LIN {X 0,Y 574.396,Z 596.267,A -85,B 0,C 180,E1 -2267.811,E2 -2267.811} C_VEL
LIN {X 0,Y 574.661,Z 582.717,A -85,B 0,C 180,E1 -2268.633,E2 -2268.633} C_VEL
LIN {X 0,Y 574.868,Z 568.152,A -85,B 0,C 180,E1 -2269.364,E2 -2269.364} C_VEL
LIN {X 0,Y 575.125,Z 552.245,A -85,B 0,C 180,E1 -2270.008,E2 -2270.008} C_VEL
LIN {X 0,Y 575.36,Z 536.014,A -85,B 0,C 180,E1 -2270.513,E2 -2270.513} C_VEL
LIN {X 0,Y 575.491,Z 519.437,A -85,B 0,C 180,E1 -2270.882,E2 -2270.882} C_VEL
LIN {X 0,Y 576.152,Z 335.908,A -85,B 0,C 180,E1 -2273.297,E2 -2273.297} C_VEL
LIN {X 0,Y 576.125,Z 317.842,A -85,B 0,C 180,E1 -2273.539,E2 -2273.539} C_VEL
LIN {X 0,Y 575.045,Z 311.76,A -85,B 0,C 180,E1 -2273.688,E2 -2273.688} C_VEL
LIN {X 0,Y 575.605,Z 275.988,A -85,B 0,C 180,E1 -2276.796,E2 -2276.796} C_VEL
LIN {X 0,Y 575.443,Z 270.866,A -85,B 0,C 180,E1 -2277.257,E2 -2277.257} C_VEL
LIN {X 0,Y 573.255,Z 263.39,A -85,B 0,C 180,E1 -2278.04,E2 -2278.04} C_VEL
LIN {X 0,Y 573.23,Z 263.394,A -85,B 0,C 180,E1 -2280.883,E2 -2280.883} C_VEL
LIN {X 0,Y 573.26,Z 263.392,A -85,B 0,C 180,E1 -2283.524,E2 -2283.524} C_VEL
LIN {X 0,Y 573.213,Z 263.391,A -85,B 0,C 180,E1 -2286.051,E2 -2286.051} C_VEL
LIN {X 0,Y 573.245,Z 263.388,A -85,B 0,C 180,E1 -2288.701,E2 -2288.701} C_VEL
LIN {X 0,Y 573.251,Z 263.39,A -85,B 0,C 180,E1 -2291.595,E2 -2291.595} C_VEL
LIN {X 0,Y 573.237,Z 263.387,A -85,B 0,C 180,E1 -2294.333,E2 -2294.333} C_VEL
LIN {X 0,Y 573.237,Z 263.394,A -85,B 0,C 180,E1 -2297.358,E2 -2297.358} C_VEL
LIN {X 0,Y 573.272,Z 263.388,A -85,B 0,C 180,E1 -2299.477,E2 -2299.477} C_VEL
LIN {X 0,Y 573.233,Z 263.387,A -85,B 0,C 180,E1 -2302.192,E2 -2302.192} C_VEL
LIN {X 0,Y 573.253,Z 263.388,A -85,B 0,C 180,E1 -2304.816,E2 -2304.816} C_VEL
LIN {X 0,Y 573.25,Z 263.393,A -85,B 0,C 180,E1 -2307.355,E2 -2307.355} C_VEL
LIN {X 0,Y 573.245,Z 263.386,A -85,B 0,C 180,E1 -2310.512,E2 -2310.512} C_VEL
LIN {X 0,Y 573.247,Z 263.393,A -85,B 0,C 180,E1 -2313.024,E2 -2313.024} C_VEL
LIN {X 0,Y 573.272,Z 263.389,A -85,B 0,C 180,E1 -2315.366,E2 -2315.366} C_VEL
LIN {X 0,Y 573.226,Z 263.389,A -85,B 0,C 180,E1 -2318.419,E2 -2318.419} C_VEL
LIN {X 0,Y 573.266,Z 263.383,A -85,B 0,C 180,E1 -2320.731,E2 -2320.731} C_VEL
LIN {X 0,Y 573.248,Z 263.388,A -85,B 0,C 180,E1 -2323.622,E2 -2323.622} C_VEL
LIN {X 0,Y 573.27,Z 263.38,A -85,B 0,C 180,E1 -2325.807,E2 -2325.807} C_VEL
LIN {X 0,Y 573.26,Z 263.387,A -85,B 0,C 180,E1 -2328.745,E2 -2328.745} C_VEL
LIN {X 0,Y 573.282,Z 263.383,A -85,B 0,C 180,E1 -2331.541,E2 -2331.541} C_VEL
LIN {X 0,Y 573.295,Z 263.377,A -85,B 0,C 180,E1 -2334.372,E2 -2334.372} C_VEL
LIN {X 0,Y 573.312,Z 263.378,A -85,B 0,C 180,E1 -2337.893,E2 -2337.893} C_VEL
LIN {X 0,Y 573.327,Z 263.377,A -85,B 0,C 180,E1 -2340.702,E2 -2340.702} C_VEL
LIN {X 0,Y 573.302,Z 263.383,A -85,B 0,C 180,E1 -2342.811,E2 -2342.811} C_VEL
LIN {X 0,Y 573.295,Z 263.38,A -85,B 0,C 180,E1 -2345.628,E2 -2345.628} C_VEL
LIN {X 0,Y 573.282,Z 263.379,A -85,B 0,C 180,E1 -2348.46,E2 -2348.46} C_VEL
LIN {X 0,Y 573.27,Z 263.388,A -85,B 0,C 180,E1 -2351.312,E2 -2351.312} C_VEL
LIN {X 0,Y 573.28,Z 263.382,A -85,B 0,C 180,E1 -2354.425,E2 -2354.425} C_VEL
LIN {X 0,Y 573.256,Z 263.392,A -85,B 0,C 180,E1 -2357.112,E2 -2357.112} C_VEL
LIN {X 0,Y 573.249,Z 263.385,A -85,B 0,C 180,E1 -2360.077,E2 -2360.077} C_VEL
LIN {X 0,Y 573.232,Z 263.395,A -85,B 0,C 180,E1 -2363.1,E2 -2363.1} C_VEL
LIN {X 0,Y 573.248,Z 263.387,A -85,B 0,C 180,E1 -2364.383,E2 -2364.383} C_VEL
LIN {X 0,Y 572.621,Z 263.473,A -85,B 0,C 180,E1 -2364.97,E2 -2364.97} C_VEL
LIN {X 0,Y 569.779,Z 263.826,A -85,B 0,C 180,E1 -2365.921,E2 -2365.921} C_VEL
LIN {X 0,Y 567.347,Z 264.127,A -85,B 0,C 180,E1 -2366.686,E2 -2366.686} C_VEL
LIN {X 0,Y 566.292,Z 264.253,A -85,B 0,C 180,E1 -2367.277,E2 -2367.277} C_VEL
LIN {X 0,Y 566.201,Z 264.261,A -85,B 0,C 180,E1 -2367.478,E2 -2367.478} C_VEL
LIN {X 0,Y 566.199,Z 264.264,A -85,B 0,C 180,E1 -2369.769,E2 -2369.769} C_VEL
LIN {X 0,Y 566.201,Z 264.266,A -85,B 0,C 180,E1 -2372.43,E2 -2372.43} C_VEL
LIN {X 0,Y 566.212,Z 264.27,A -85,B 0,C 180,E1 -2374.995,E2 -2374.995} C_VEL
LIN {X 0,Y 566.195,Z 264.263,A -85,B 0,C 180,E1 -2377.461,E2 -2377.461} C_VEL
LIN {X 0,Y 566.206,Z 264.264,A -85,B 0,C 180,E1 -2380.199,E2 -2380.199} C_VEL
LIN {X 0,Y 566.2,Z 264.27,A -85,B 0,C 180,E1 -2383.054,E2 -2383.054} C_VEL
LIN {X 0,Y 566.201,Z 264.262,A -85,B 0,C 180,E1 -2386.049,E2 -2386.049} C_VEL
LIN {X 0,Y 566.211,Z 264.272,A -85,B 0,C 180,E1 -2388.864,E2 -2388.864} C_VEL
LIN {X 0,Y 566.188,Z 264.264,A -85,B 0,C 180,E1 -2391.637,E2 -2391.637} C_VEL
LIN {X 0,Y 566.161,Z 264.27,A -85,B 0,C 180,E1 -2394.308,E2 -2394.308} C_VEL
LIN {X 0,Y 566.219,Z 264.266,A -85,B 0,C 180,E1 -2396.898,E2 -2396.898} C_VEL
LIN {X 0,Y 566.183,Z 264.269,A -85,B 0,C 180,E1 -2399.408,E2 -2399.408} C_VEL
LIN {X 0,Y 566.212,Z 264.265,A -85,B 0,C 180,E1 -2401.858,E2 -2401.858} C_VEL
LIN {X 0,Y 566.254,Z 264.454,A -85,B 0,C 180,E1 -2404.13,E2 -2404.13} C_VEL
LIN {X 0,Y 568.203,Z 272.217,A -85,B 0,C 180,E1 -2405.022,E2 -2405.022} C_VEL
LIN {X 0,Y 568.08,Z 282.889,A -85,B 0,C 180,E1 -2406.085,E2 -2406.085} C_VEL
LIN {X 0,Y 569.697,Z 291.686,A -85,B 0,C 180,E1 -2406.276,E2 -2406.276} C_VEL
LIN {X 0,Y 568.883,Z 488.854,A -85,B 0,C 180,E1 -2408.9,E2 -2408.9} C_VEL
LIN {X 0,Y 568.716,Z 505.193,A -85,B 0,C 180,E1 -2409.26,E2 -2409.26} C_VEL
LIN {X 0,Y 568.457,Z 521.005,A -85,B 0,C 180,E1 -2409.747,E2 -2409.747} C_VEL
LIN {X 0,Y 568.168,Z 537.348,A -85,B 0,C 180,E1 -2410.405,E2 -2410.405} C_VEL
LIN {X 0,Y 567.887,Z 551.932,A -85,B 0,C 180,E1 -2411.137,E2 -2411.137} C_VEL
LIN {X 0,Y 567.549,Z 566.935,A -85,B 0,C 180,E1 -2412.055,E2 -2412.055} C_VEL
LIN {X 0,Y 567.21,Z 580.823,A -85,B 0,C 180,E1 -2413.072,E2 -2413.072} C_VEL
LIN {X 0,Y 566.947,Z 593.594,A -85,B 0,C 180,E1 -2414.174,E2 -2414.174} C_VEL
LIN {X 0,Y 566.624,Z 605.25,A -85,B 0,C 180,E1 -2415.342,E2 -2415.342} C_VEL
LIN {X 0,Y 566.435,Z 617.002,A -85,B 0,C 180,E1 -2416.73,E2 -2416.73} C_VEL
LIN {X 0,Y 566.241,Z 627.369,A -85,B 0,C 180,E1 -2418.183,E2 -2418.183} C_VEL
LIN {X 0,Y 566.133,Z 636.034,A -85,B 0,C 180,E1 -2419.63,E2 -2419.63} C_VEL
LIN {X 0,Y 566.012,Z 643.287,A -85,B 0,C 180,E1 -2421.071,E2 -2421.071} C_VEL
LIN {X 0,Y 565.97,Z 649.294,A -85,B 0,C 180,E1 -2422.508,E2 -2422.508} C_VEL
LIN {X 0,Y 565.915,Z 654.055,A -85,B 0,C 180,E1 -2423.941,E2 -2423.941} C_VEL
LIN {X 0,Y 565.913,Z 658.544,A -85,B 0,C 180,E1 -2425.727,E2 -2425.727} C_VEL
LIN {X 0,Y 565.866,Z 661.021,A -85,B 0,C 180,E1 -2427.152,E2 -2427.152} C_VEL
LIN {X 0,Y 565.84,Z 662.45,A -85,B 0,C 180,E1 -2428.577,E2 -2428.577} C_VEL
LIN {X 0,Y 565.835,Z 662.996,A -85,B 0,C 180,E1 -2430,E2 -2430} C_VEL
LIN {X 0,Y 565.838,Z 662.509,A -85,B 0,C 180,E1 -2431.423,E2 -2431.423} C_VEL
LIN {X 0,Y 565.867,Z 661.149,A -85,B 0,C 180,E1 -2432.848,E2 -2432.848} C_VEL
LIN {X 0,Y 565.91,Z 658.728,A -85,B 0,C 180,E1 -2434.273,E2 -2434.273} C_VEL
LIN {X 0,Y 565.964,Z 655.378,A -85,B 0,C 180,E1 -2435.701,E2 -2435.701} C_VEL
LIN {X 0,Y 565.967,Z 650.873,A -85,B 0,C 180,E1 -2437.133,E2 -2437.133} C_VEL
LIN {X 0,Y 566.022,Z 645.304,A -85,B 0,C 180,E1 -2438.569,E2 -2438.569} C_VEL
LIN {X 0,Y 566.084,Z 638.461,A -85,B 0,C 180,E1 -2440.009,E2 -2440.009} C_VEL
LIN {X 0,Y 566.209,Z 630.214,A -85,B 0,C 180,E1 -2441.455,E2 -2441.455} C_VEL
LIN {X 0,Y 566.363,Z 620.389,A -85,B 0,C 180,E1 -2442.906,E2 -2442.906} C_VEL
LIN {X 0,Y 566.58,Z 610.288,A -85,B 0,C 180,E1 -2444.181,E2 -2444.181} C_VEL
LIN {X 0,Y 566.797,Z 598.38,A -85,B 0,C 180,E1 -2445.461,E2 -2445.461} C_VEL
LIN {X 0,Y 567.124,Z 585.297,A -85,B 0,C 180,E1 -2446.653,E2 -2446.653} C_VEL
LIN {X 0,Y 567.419,Z 572.581,A -85,B 0,C 180,E1 -2447.641,E2 -2447.641} C_VEL
LIN {X 0,Y 567.757,Z 558.218,A -85,B 0,C 180,E1 -2448.587,E2 -2448.587} C_VEL
LIN {X 0,Y 568.074,Z 543.006,A -85,B 0,C 180,E1 -2449.42,E2 -2449.42} C_VEL
LIN {X 0,Y 568.353,Z 528.125,A -85,B 0,C 180,E1 -2450.077,E2 -2450.077} C_VEL
LIN {X 0,Y 568.613,Z 512.384,A -85,B 0,C 180,E1 -2450.625,E2 -2450.625} C_VEL
LIN {X 0,Y 568.809,Z 495.094,A -85,B 0,C 180,E1 -2451.068,E2 -2451.068} C_VEL
LIN {X 0,Y 568.982,Z 478.408,A -85,B 0,C 180,E1 -2451.345,E2 -2451.345} C_VEL
LIN {X 0,Y 569.679,Z 290.701,A -85,B 0,C 180,E1 -2453.828,E2 -2453.828} C_VEL
LIN {X 0,Y 568.068,Z 282.675,A -85,B 0,C 180,E1 -2454.027,E2 -2454.027} C_VEL
LIN {X 0,Y 568.089,Z 271.64,A -85,B 0,C 180,E1 -2455.133,E2 -2455.133} C_VEL
LIN {X 0,Y 566.221,Z 264.268,A -85,B 0,C 180,E1 -2455.995,E2 -2455.995} C_VEL
LIN {X 0,Y 566.186,Z 264.272,A -85,B 0,C 180,E1 -2458.953,E2 -2458.953} C_VEL
LIN {X 0,Y 566.191,Z 264.274,A -85,B 0,C 180,E1 -2461.422,E2 -2461.422} C_VEL
LIN {X 0,Y 566.208,Z 264.266,A -85,B 0,C 180,E1 -2463.956,E2 -2463.956} C_VEL
LIN {X 0,Y 566.181,Z 264.264,A -85,B 0,C 180,E1 -2466.571,E2 -2466.571} C_VEL
LIN {X 0,Y 566.213,Z 264.266,A -85,B 0,C 180,E1 -2469.685,E2 -2469.685} C_VEL
LIN {X 0,Y 566.203,Z 264.267,A -85,B 0,C 180,E1 -2472.917,E2 -2472.917} C_VEL
LIN {X 0,Y 566.197,Z 264.264,A -85,B 0,C 180,E1 -2476.048,E2 -2476.048} C_VEL
LIN {X 0,Y 566.177,Z 264.27,A -85,B 0,C 180,E1 -2478.861,E2 -2478.861} C_VEL
LIN {X 0,Y 566.184,Z 264.268,A -85,B 0,C 180,E1 -2481.637,E2 -2481.637} C_VEL
LIN {X 0,Y 566.195,Z 264.264,A -85,B 0,C 180,E1 -2484.31,E2 -2484.31} C_VEL
LIN {X 0,Y 566.217,Z 264.266,A -85,B 0,C 180,E1 -2486.898,E2 -2486.898} C_VEL
LIN {X 0,Y 566.179,Z 264.272,A -85,B 0,C 180,E1 -2489.407,E2 -2489.407} C_VEL
LIN {X 0,Y 566.209,Z 264.26,A -85,B 0,C 180,E1 -2491.857,E2 -2491.857} C_VEL
LIN {X 0,Y 566.21,Z 264.262,A -85,B 0,C 180,E1 -2494.251,E2 -2494.251} C_VEL
LIN {X 0,Y 566.189,Z 264.268,A -85,B 0,C 180,E1 -2496.714,E2 -2496.714} C_VEL
LIN {X 0,Y 566.206,Z 264.265,A -85,B 0,C 180,E1 -2499.662,E2 -2499.662} C_VEL
LIN {X 0,Y 566.197,Z 264.267,A -85,B 0,C 180,E1 -2502.668,E2 -2502.668} C_VEL
LIN {X 0,Y 566.232,Z 264.261,A -85,B 0,C 180,E1 -2505.627,E2 -2505.627} C_VEL
LIN {X 0,Y 566.232,Z 264.263,A -85,B 0,C 180,E1 -2508.675,E2 -2508.675} C_VEL
LIN {X 0,Y 566.225,Z 264.263,A -85,B 0,C 180,E1 -2511.434,E2 -2511.434} C_VEL
LIN {X 0,Y 566.265,Z 264.256,A -85,B 0,C 180,E1 -2514.302,E2 -2514.302} C_VEL
LIN {X 0,Y 566.282,Z 264.25,A -85,B 0,C 180,E1 -2517.866,E2 -2517.866} C_VEL
LIN {X 0,Y 566.299,Z 264.257,A -85,B 0,C 180,E1 -2520.711,E2 -2520.711} C_VEL
LIN {X 0,Y 566.269,Z 264.262,A -85,B 0,C 180,E1 -2522.845,E2 -2522.845} C_VEL
LIN {X 0,Y 566.265,Z 264.256,A -85,B 0,C 180,E1 -2525.698,E2 -2525.698} C_VEL
LIN {X 0,Y 566.225,Z 264.264,A -85,B 0,C 180,E1 -2528.566,E2 -2528.566} C_VEL
LIN {X 0,Y 566.239,Z 264.26,A -85,B 0,C 180,E1 -2531.454,E2 -2531.454} C_VEL
LIN {X 0,Y 566.231,Z 264.263,A -85,B 0,C 180,E1 -2534.507,E2 -2534.507} C_VEL
LIN {X 0,Y 566.197,Z 264.267,A -85,B 0,C 180,E1 -2537.332,E2 -2537.332} C_VEL
LIN {X 0,Y 566.21,Z 264.265,A -85,B 0,C 180,E1 -2540.337,E2 -2540.337} C_VEL
LIN {X 0,Y 566.186,Z 264.268,A -85,B 0,C 180,E1 -2543.404,E2 -2543.404} C_VEL
LIN {X 0,Y 566.209,Z 264.263,A -85,B 0,C 180,E1 -2545.749,E2 -2545.749} C_VEL
LIN {X 0,Y 566.199,Z 264.266,A -85,B 0,C 180,E1 -2548.202,E2 -2548.202} C_VEL
LIN {X 0,Y 566.188,Z 264.272,A -85,B 0,C 180,E1 -2551.077,E2 -2551.077} C_VEL
LIN {X 0,Y 566.209,Z 264.264,A -85,B 0,C 180,E1 -2553.734,E2 -2553.734} C_VEL
LIN {X 0,Y 566.213,Z 264.269,A -85,B 0,C 180,E1 -2556.569,E2 -2556.569} C_VEL
LIN {X 0,Y 566.204,Z 264.264,A -85,B 0,C 180,E1 -2559.685,E2 -2559.685} C_VEL
LIN {X 0,Y 566.21,Z 264.265,A -85,B 0,C 180,E1 -2562.087,E2 -2562.087} C_VEL
LIN {X 0,Y 566.171,Z 264.273,A -85,B 0,C 180,E1 -2565.036,E2 -2565.036} C_VEL
LIN {X 0,Y 566.216,Z 264.264,A -85,B 0,C 180,E1 -2568.136,E2 -2568.136} C_VEL
LIN {X 0,Y 566.217,Z 264.271,A -85,B 0,C 180,E1 -2570.727,E2 -2570.727} C_VEL
LIN {X 0,Y 566.182,Z 264.267,A -85,B 0,C 180,E1 -2573.788,E2 -2573.788} C_VEL
LIN {X 0,Y 566.209,Z 264.264,A -85,B 0,C 180,E1 -2576.266,E2 -2576.266} C_VEL
LIN {X 0,Y 566.191,Z 264.273,A -85,B 0,C 180,E1 -2578.923,E2 -2578.923} C_VEL
LIN {X 0,Y 566.24,Z 264.409,A -85,B 0,C 180,E1 -2581.703,E2 -2581.703} C_VEL
LIN {X 0,Y 568.798,Z 273.135,A -85,B 0,C 180,E1 -2582.617,E2 -2582.617} C_VEL
LIN {X 0,Y 568.763,Z 287.404,A -85,B 0,C 180,E1 -2583.883,E2 -2583.883} C_VEL
LIN {X 0,Y 568.329,Z 311.996,A -85,B 0,C 180,E1 -2586.036,E2 -2586.036} C_VEL
LIN {X 0,Y 569.734,Z 319.846,A -85,B 0,C 180,E1 -2586.208,E2 -2586.208} C_VEL
LIN {X 0,Y 568.873,Z 519.439,A -85,B 0,C 180,E1 -2588.864,E2 -2588.864} C_VEL
LIN {X 0,Y 568.726,Z 536.014,A -85,B 0,C 180,E1 -2589.237,E2 -2589.237} C_VEL
LIN {X 0,Y 568.422,Z 552.246,A -85,B 0,C 180,E1 -2589.746,E2 -2589.746} C_VEL
LIN {X 0,Y 568.148,Z 568.383,A -85,B 0,C 180,E1 -2590.408,E2 -2590.408} C_VEL
LIN {X 0,Y 567.878,Z 582.718,A -85,B 0,C 180,E1 -2591.136,E2 -2591.136} C_VEL
LIN {X 0,Y 567.582,Z 596.271,A -85,B 0,C 180,E1 -2591.968,E2 -2591.968} C_VEL
LIN {X 0,Y 567.228,Z 610.22,A -85,B 0,C 180,E1 -2592.98,E2 -2592.98} C_VEL
LIN {X 0,Y 566.915,Z 624.071,A -85,B 0,C 180,E1 -2594.173,E2 -2594.173} C_VEL
LIN {X 0,Y 566.63,Z 635.62,A -85,B 0,C 180,E1 -2595.339,E2 -2595.339} C_VEL
LIN {X 0,Y 566.434,Z 647.338,A -85,B 0,C 180,E1 -2596.73,E2 -2596.73} C_VEL
LIN {X 0,Y 566.238,Z 657.673,A -85,B 0,C 180,E1 -2598.183,E2 -2598.183} C_VEL
LIN {X 0,Y 566.12,Z 666.285,A -85,B 0,C 180,E1 -2599.63,E2 -2599.63} C_VEL
LIN {X 0,Y 566.001,Z 673.489,A -85,B 0,C 180,E1 -2601.071,E2 -2601.071} C_VEL
LIN {X 0,Y 565.968,Z 679.467,A -85,B 0,C 180,E1 -2602.508,E2 -2602.508} C_VEL
LIN {X 0,Y 565.915,Z 684.187,A -85,B 0,C 180,E1 -2603.941,E2 -2603.941} C_VEL
LIN {X 0,Y 565.911,Z 688.637,A -85,B 0,C 180,E1 -2605.727,E2 -2605.727} C_VEL
LIN {X 0,Y 565.866,Z 691.089,A -85,B 0,C 180,E1 -2607.152,E2 -2607.152} C_VEL
LIN {X 0,Y 565.839,Z 692.48,A -85,B 0,C 180,E1 -2608.577,E2 -2608.577} C_VEL
LIN {X 0,Y 565.834,Z 693,A -85,B 0,C 180,E1 -2610,E2 -2610} C_VEL
LIN {X 0,Y 565.839,Z 692.48,A -85,B 0,C 180,E1 -2611.423,E2 -2611.423} C_VEL
LIN {X 0,Y 565.866,Z 691.088,A -85,B 0,C 180,E1 -2612.848,E2 -2612.848} C_VEL
LIN {X 0,Y 565.911,Z 688.636,A -85,B 0,C 180,E1 -2614.273,E2 -2614.273} C_VEL
LIN {X 0,Y 565.914,Z 684.188,A -85,B 0,C 180,E1 -2616.059,E2 -2616.059} C_VEL
LIN {X 0,Y 565.968,Z 679.468,A -85,B 0,C 180,E1 -2617.492,E2 -2617.492} C_VEL
LIN {X 0,Y 566.001,Z 673.489,A -85,B 0,C 180,E1 -2618.929,E2 -2618.929} C_VEL
LIN {X 0,Y 566.126,Z 665.277,A -85,B 0,C 180,E1 -2620.551,E2 -2620.551} C_VEL
LIN {X 0,Y 566.246,Z 656.443,A -85,B 0,C 180,E1 -2621.999,E2 -2621.999} C_VEL
LIN {X 0,Y 566.427,Z 645.908,A -85,B 0,C 180,E1 -2623.453,E2 -2623.453} C_VEL
LIN {X 0,Y 566.66,Z 634.612,A -85,B 0,C 180,E1 -2624.773,E2 -2624.773} C_VEL
LIN {X 0,Y 566.957,Z 622.119,A -85,B 0,C 180,E1 -2626.01,E2 -2626.01} C_VEL
LIN {X 0,Y 567.229,Z 609.046,A -85,B 0,C 180,E1 -2627.113,E2 -2627.113} C_VEL
LIN {X 0,Y 567.6,Z 594.852,A -85,B 0,C 180,E1 -2628.125,E2 -2628.125} C_VEL
LIN {X 0,Y 567.9,Z 581.028,A -85,B 0,C 180,E1 -2628.957,E2 -2628.957} C_VEL
LIN {X 0,Y 568.196,Z 566.527,A -85,B 0,C 180,E1 -2629.678,E2 -2629.678} C_VEL
LIN {X 0,Y 568.444,Z 550.945,A -85,B 0,C 180,E1 -2630.301,E2 -2630.301} C_VEL
LIN {X 0,Y 568.734,Z 534.187,A -85,B 0,C 180,E1 -2630.81,E2 -2630.81} C_VEL
LIN {X 0,Y 568.889,Z 517.947,A -85,B 0,C 180,E1 -2631.159,E2 -2631.159} C_VEL
LIN {X 0,Y 569.679,Z 320.023,A -85,B 0,C 180,E1 -2633.792,E2 -2633.792} C_VEL
LIN {X 0,Y 568.354,Z 311.826,A -85,B 0,C 180,E1 -2633.978,E2 -2633.978} C_VEL
LIN {X 0,Y 568.942,Z 276.869,A -85,B 0,C 180,E1 -2637.043,E2 -2637.043} C_VEL
LIN {X 0,Y 568.734,Z 272.912,A -85,B 0,C 180,E1 -2637.406,E2 -2637.406} C_VEL
LIN {X 0,Y 566.216,Z 264.266,A -85,B 0,C 180,E1 -2638.324,E2 -2638.324} C_VEL
LIN {X 0,Y 566.193,Z 264.273,A -85,B 0,C 180,E1 -2641.422,E2 -2641.422} C_VEL
LIN {X 0,Y 566.207,Z 264.266,A -85,B 0,C 180,E1 -2643.956,E2 -2643.956} C_VEL
LIN {X 0,Y 566.198,Z 264.266,A -85,B 0,C 180,E1 -2646.57,E2 -2646.57} C_VEL
LIN {X 0,Y 566.218,Z 264.266,A -85,B 0,C 180,E1 -2649.686,E2 -2649.686} C_VEL
LIN {X 0,Y 566.211,Z 264.263,A -85,B 0,C 180,E1 -2652.087,E2 -2652.087} C_VEL
LIN {X 0,Y 566.171,Z 264.273,A -85,B 0,C 180,E1 -2655.036,E2 -2655.036} C_VEL
LIN {X 0,Y 566.215,Z 264.261,A -85,B 0,C 180,E1 -2658.136,E2 -2658.136} C_VEL
LIN {X 0,Y 566.213,Z 264.263,A -85,B 0,C 180,E1 -2660.726,E2 -2660.726} C_VEL
LIN {X 0,Y 566.204,Z 264.264,A -85,B 0,C 180,E1 -2663.785,E2 -2663.785} C_VEL
LIN {X 0,Y 566.209,Z 264.262,A -85,B 0,C 180,E1 -2666.266,E2 -2666.266} C_VEL
LIN {X 0,Y 566.188,Z 264.27,A -85,B 0,C 180,E1 -2668.923,E2 -2668.923} C_VEL
LIN {X 0,Y 566.208,Z 264.263,A -85,B 0,C 180,E1 -2671.857,E2 -2671.857} C_VEL
LIN {X 0,Y 566.21,Z 264.263,A -85,B 0,C 180,E1 -2674.251,E2 -2674.251} C_VEL
LIN {X 0,Y 566.189,Z 264.268,A -85,B 0,C 180,E1 -2676.714,E2 -2676.714} C_VEL
LIN {X 0,Y 566.206,Z 264.261,A -85,B 0,C 180,E1 -2679.663,E2 -2679.663} C_VEL
LIN {X 0,Y 566.197,Z 264.267,A -85,B 0,C 180,E1 -2682.668,E2 -2682.668} C_VEL
LIN {X 0,Y 566.231,Z 264.258,A -85,B 0,C 180,E1 -2685.627,E2 -2685.627} C_VEL
LIN {X 0,Y 566.232,Z 264.262,A -85,B 0,C 180,E1 -2688.675,E2 -2688.675} C_VEL
LIN {X 0,Y 566.225,Z 264.263,A -85,B 0,C 180,E1 -2691.434,E2 -2691.434} C_VEL
LIN {X 0,Y 566.264,Z 264.252,A -85,B 0,C 180,E1 -2694.302,E2 -2694.302} C_VEL
LIN {X 0,Y 566.283,Z 264.253,A -85,B 0,C 180,E1 -2697.866,E2 -2697.866} C_VEL
LIN {X 0,Y 566.298,Z 264.252,A -85,B 0,C 180,E1 -2700.711,E2 -2700.711} C_VEL
LIN {X 0,Y 566.269,Z 264.259,A -85,B 0,C 180,E1 -2702.846,E2 -2702.846} C_VEL
LIN {X 0,Y 566.262,Z 264.256,A -85,B 0,C 180,E1 -2705.698,E2 -2705.698} C_VEL
LIN {X 0,Y 566.226,Z 264.258,A -85,B 0,C 180,E1 -2708.566,E2 -2708.566} C_VEL
LIN {X 0,Y 566.24,Z 264.262,A -85,B 0,C 180,E1 -2711.454,E2 -2711.454} C_VEL
LIN {X 0,Y 566.232,Z 264.26,A -85,B 0,C 180,E1 -2714.507,E2 -2714.507} C_VEL
LIN {X 0,Y 566.198,Z 264.268,A -85,B 0,C 180,E1 -2717.332,E2 -2717.332} C_VEL
LIN {X 0,Y 566.211,Z 264.263,A -85,B 0,C 180,E1 -2720.337,E2 -2720.337} C_VEL
LIN {X 0,Y 566.188,Z 264.268,A -85,B 0,C 180,E1 -2723.404,E2 -2723.404} C_VEL
LIN {X 0,Y 566.211,Z 264.262,A -85,B 0,C 180,E1 -2725.749,E2 -2725.749} C_VEL
LIN {X 0,Y 566.201,Z 264.261,A -85,B 0,C 180,E1 -2727.478,E2 -2727.478} C_VEL
LIN {X 0,Y 565.521,Z 264.347,A -85,B 0,C 180,E1 -2728.071,E2 -2728.071} C_VEL
LIN {X 0,Y 562.655,Z 264.713,A -85,B 0,C 180,E1 -2729.035,E2 -2729.035} C_VEL
LIN {X 0,Y 560.246,Z 265.009,A -85,B 0,C 180,E1 -2729.811,E2 -2729.811} C_VEL
LIN {X 0,Y 559.218,Z 265.136,A -85,B 0,C 180,E1 -2730.409,E2 -2730.409} C_VEL
LIN {X 0,Y 559.138,Z 265.146,A -85,B 0,C 180,E1 -2730.612,E2 -2730.612} C_VEL
LIN {X 0,Y 559.161,Z 265.141,A -85,B 0,C 180,E1 -2733.575,E2 -2733.575} C_VEL
LIN {X 0,Y 559.168,Z 265.143,A -85,B 0,C 180,E1 -2736.449,E2 -2736.449} C_VEL
LIN {X 0,Y 559.173,Z 265.146,A -85,B 0,C 180,E1 -2738.934,E2 -2738.934} C_VEL
LIN {X 0,Y 559.173,Z 265.138,A -85,B 0,C 180,E1 -2742.137,E2 -2742.137} C_VEL
LIN {X 0,Y 559.139,Z 265.144,A -85,B 0,C 180,E1 -2745.261,E2 -2745.261} C_VEL
LIN {X 0,Y 559.191,Z 265.139,A -85,B 0,C 180,E1 -2748.233,E2 -2748.233} C_VEL
LIN {X 0,Y 559.177,Z 265.141,A -85,B 0,C 180,E1 -2751.192,E2 -2751.192} C_VEL
LIN {X 0,Y 559.138,Z 265.142,A -85,B 0,C 180,E1 -2753.789,E2 -2753.789} C_VEL
LIN {X 0,Y 559.162,Z 265.145,A -85,B 0,C 180,E1 -2756.425,E2 -2756.425} C_VEL
LIN {X 0,Y 559.158,Z 265.148,A -85,B 0,C 180,E1 -2758.981,E2 -2758.981} C_VEL
LIN {X 0,Y 559.145,Z 265.146,A -85,B 0,C 180,E1 -2761.623,E2 -2761.623} C_VEL
LIN {X 0,Y 559.215,Z 265.248,A -85,B 0,C 180,E1 -2763.842,E2 -2763.842} C_VEL
LIN {X 0,Y 561.348,Z 273.487,A -85,B 0,C 180,E1 -2764.807,E2 -2764.807} C_VEL
LIN {X 0,Y 561.457,Z 279.258,A -85,B 0,C 180,E1 -2765.405,E2 -2765.405} C_VEL
LIN {X 0,Y 561.412,Z 283.277,A -85,B 0,C 180,E1 -2765.787,E2 -2765.787} C_VEL
LIN {X 0,Y 563.205,Z 292.276,A -85,B 0,C 180,E1 -2765.993,E2 -2765.993} C_VEL
LIN {X 0,Y 562.264,Z 488.139,A -85,B 0,C 180,E1 -2768.627,E2 -2768.627} C_VEL
LIN {X 0,Y 562.067,Z 504.3,A -85,B 0,C 180,E1 -2768.98,E2 -2768.98} C_VEL
LIN {X 0,Y 561.78,Z 521.02,A -85,B 0,C 180,E1 -2769.495,E2 -2769.495} C_VEL
LIN {X 0,Y 561.495,Z 535.996,A -85,B 0,C 180,E1 -2770.097,E2 -2770.097} C_VEL
LIN {X 0,Y 561.15,Z 550.204,A -85,B 0,C 180,E1 -2770.806,E2 -2770.806} C_VEL
LIN {X 0,Y 560.804,Z 564.169,A -85,B 0,C 180,E1 -2771.647,E2 -2771.647} C_VEL
LIN {X 0,Y 560.391,Z 578.482,A -85,B 0,C 180,E1 -2772.671,E2 -2772.671} C_VEL
LIN {X 0,Y 559.991,Z 591.648,A -85,B 0,C 180,E1 -2773.785,E2 -2773.785} C_VEL
LIN {X 0,Y 559.698,Z 604.552,A -85,B 0,C 180,E1 -2775.077,E2 -2775.077} C_VEL
LIN {X 0,Y 559.451,Z 615.547,A -85,B 0,C 180,E1 -2776.376,E2 -2776.376} C_VEL
LIN {X 0,Y 559.252,Z 624.91,A -85,B 0,C 180,E1 -2777.665,E2 -2777.665} C_VEL
LIN {X 0,Y 559.068,Z 634.017,A -85,B 0,C 180,E1 -2779.131,E2 -2779.131} C_VEL
LIN {X 0,Y 558.941,Z 641.635,A -85,B 0,C 180,E1 -2780.592,E2 -2780.592} C_VEL
LIN {X 0,Y 558.892,Z 647.873,A -85,B 0,C 180,E1 -2782.049,E2 -2782.049} C_VEL
LIN {X 0,Y 558.818,Z 653.573,A -85,B 0,C 180,E1 -2783.699,E2 -2783.699} C_VEL
LIN {X 0,Y 558.777,Z 656.95,A -85,B 0,C 180,E1 -2784.949,E2 -2784.949} C_VEL
LIN {X 0,Y 558.817,Z 659.909,A -85,B 0,C 180,E1 -2786.395,E2 -2786.395} C_VEL
LIN {X 0,Y 558.741,Z 661.845,A -85,B 0,C 180,E1 -2787.837,E2 -2787.837} C_VEL
LIN {X 0,Y 558.736,Z 662.839,A -85,B 0,C 180,E1 -2789.279,E2 -2789.279} C_VEL
LIN {X 0,Y 558.736,Z 662.859,A -85,B 0,C 180,E1 -2790.721,E2 -2790.721} C_VEL
LIN {X 0,Y 558.742,Z 661.943,A -85,B 0,C 180,E1 -2792.163,E2 -2792.163} C_VEL
LIN {X 0,Y 558.817,Z 660.05,A -85,B 0,C 180,E1 -2793.605,E2 -2793.605} C_VEL
LIN {X 0,Y 558.775,Z 657.17,A -85,B 0,C 180,E1 -2795.051,E2 -2795.051} C_VEL
LIN {X 0,Y 558.843,Z 653.146,A -85,B 0,C 180,E1 -2796.535,E2 -2796.535} C_VEL
LIN {X 0,Y 558.892,Z 648.224,A -85,B 0,C 180,E1 -2797.951,E2 -2797.951} C_VEL
LIN {X 0,Y 558.928,Z 642.069,A -85,B 0,C 180,E1 -2799.408,E2 -2799.408} C_VEL
LIN {X 0,Y 559.052,Z 634.515,A -85,B 0,C 180,E1 -2800.869,E2 -2800.869} C_VEL
LIN {X 0,Y 559.242,Z 625.511,A -85,B 0,C 180,E1 -2802.336,E2 -2802.336} C_VEL
LIN {X 0,Y 559.465,Z 614.783,A -85,B 0,C 180,E1 -2803.808,E2 -2803.808} C_VEL
LIN {X 0,Y 559.765,Z 603.556,A -85,B 0,C 180,E1 -2805.118,E2 -2805.118} C_VEL
LIN {X 0,Y 560.078,Z 590.615,A -85,B 0,C 180,E1 -2806.399,E2 -2806.399} C_VEL
LIN {X 0,Y 560.418,Z 577.258,A -85,B 0,C 180,E1 -2807.516,E2 -2807.516} C_VEL
LIN {X 0,Y 560.809,Z 564.102,A -85,B 0,C 180,E1 -2808.447,E2 -2808.447} C_VEL
LIN {X 0,Y 561.147,Z 550.118,A -85,B 0,C 180,E1 -2809.289,E2 -2809.289} C_VEL
LIN {X 0,Y 561.519,Z 534.275,A -85,B 0,C 180,E1 -2810.071,E2 -2810.071} C_VEL
LIN {X 0,Y 561.893,Z 518.265,A -85,B 0,C 180,E1 -2810.692,E2 -2810.692} C_VEL
LIN {X 0,Y 562.112,Z 502.237,A -85,B 0,C 180,E1 -2811.163,E2 -2811.163} C_VEL
LIN {X 0,Y 562.285,Z 486.25,A -85,B 0,C 180,E1 -2811.492,E2 -2811.492} C_VEL
LIN {X 0,Y 563.194,Z 291.947,A -85,B 0,C 180,E1 -2814.102,E2 -2814.102} C_VEL
LIN {X 0,Y 561.359,Z 282.859,A -85,B 0,C 180,E1 -2814.322,E2 -2814.322} C_VEL
LIN {X 0,Y 561.495,Z 274.373,A -85,B 0,C 180,E1 -2815.186,E2 -2815.186} C_VEL
LIN {X 0,Y 559.174,Z 265.145,A -85,B 0,C 180,E1 -2816.273,E2 -2816.273} C_VEL
LIN {X 0,Y 559.139,Z 265.149,A -85,B 0,C 180,E1 -2819.354,E2 -2819.354} C_VEL
LIN {X 0,Y 559.163,Z 265.143,A -85,B 0,C 180,E1 -2821.863,E2 -2821.863} C_VEL
LIN {X 0,Y 559.141,Z 265.146,A -85,B 0,C 180,E1 -2824.445,E2 -2824.445} C_VEL
LIN {X 0,Y 559.133,Z 265.149,A -85,B 0,C 180,E1 -2827.639,E2 -2827.639} C_VEL
LIN {X 0,Y 559.159,Z 265.142,A -85,B 0,C 180,E1 -2829.941,E2 -2829.941} C_VEL
LIN {X 0,Y 559.158,Z 265.142,A -85,B 0,C 180,E1 -2832.743,E2 -2832.743} C_VEL
LIN {X 0,Y 559.151,Z 265.144,A -85,B 0,C 180,E1 -2835.76,E2 -2835.76} C_VEL
LIN {X 0,Y 559.182,Z 265.137,A -85,B 0,C 180,E1 -2838.231,E2 -2838.231} C_VEL
LIN {X 0,Y 559.173,Z 265.149,A -85,B 0,C 180,E1 -2841.191,E2 -2841.191} C_VEL
LIN {X 0,Y 559.159,Z 265.142,A -85,B 0,C 180,E1 -2843.791,E2 -2843.791} C_VEL
LIN {X 0,Y 559.16,Z 265.141,A -85,B 0,C 180,E1 -2846.425,E2 -2846.425} C_VEL
LIN {X 0,Y 559.153,Z 265.147,A -85,B 0,C 180,E1 -2848.981,E2 -2848.981} C_VEL
LIN {X 0,Y 559.166,Z 265.139,A -85,B 0,C 180,E1 -2851.619,E2 -2851.619} C_VEL
LIN {X 0,Y 559.178,Z 265.139,A -85,B 0,C 180,E1 -2853.903,E2 -2853.903} C_VEL
LIN {X 0,Y 559.154,Z 265.143,A -85,B 0,C 180,E1 -2856.567,E2 -2856.567} C_VEL
LIN {X 0,Y 559.174,Z 265.144,A -85,B 0,C 180,E1 -2859.395,E2 -2859.395} C_VEL
LIN {X 0,Y 559.141,Z 265.144,A -85,B 0,C 180,E1 -2861.685,E2 -2861.685} C_VEL
LIN {X 0,Y 559.164,Z 265.135,A -85,B 0,C 180,E1 -2863.948,E2 -2863.948} C_VEL
LIN {X 0,Y 559.169,Z 265.139,A -85,B 0,C 180,E1 -2866.184,E2 -2866.184} C_VEL
LIN {X 0,Y 559.193,Z 265.141,A -85,B 0,C 180,E1 -2869.133,E2 -2869.133} C_VEL
LIN {X 0,Y 559.201,Z 265.134,A -85,B 0,C 180,E1 -2872.053,E2 -2872.053} C_VEL
LIN {X 0,Y 559.252,Z 265.138,A -85,B 0,C 180,E1 -2874.953,E2 -2874.953} C_VEL
LIN {X 0,Y 559.253,Z 265.126,A -85,B 0,C 180,E1 -2877.839,E2 -2877.839} C_VEL
LIN {X 0,Y 559.27,Z 265.132,A -85,B 0,C 180,E1 -2880.72,E2 -2880.72} C_VEL
LIN {X 0,Y 559.235,Z 265.138,A -85,B 0,C 180,E1 -2882.881,E2 -2882.881} C_VEL
LIN {X 0,Y 559.234,Z 265.131,A -85,B 0,C 180,E1 -2885.77,E2 -2885.77} C_VEL
LIN {X 0,Y 559.184,Z 265.143,A -85,B 0,C 180,E1 -2888.674,E2 -2888.674} C_VEL
LIN {X 0,Y 559.202,Z 265.135,A -85,B 0,C 180,E1 -2891.6,E2 -2891.6} C_VEL
LIN {X 0,Y 559.197,Z 265.141,A -85,B 0,C 180,E1 -2894.595,E2 -2894.595} C_VEL
LIN {X 0,Y 559.156,Z 265.142,A -85,B 0,C 180,E1 -2897.557,E2 -2897.557} C_VEL
LIN {X 0,Y 559.169,Z 265.14,A -85,B 0,C 180,E1 -2899.837,E2 -2899.837} C_VEL
LIN {X 0,Y 559.138,Z 265.144,A -85,B 0,C 180,E1 -2902.153,E2 -2902.153} C_VEL
LIN {X 0,Y 559.176,Z 265.144,A -85,B 0,C 180,E1 -2905.187,E2 -2905.187} C_VEL
LIN {X 0,Y 559.153,Z 265.142,A -85,B 0,C 180,E1 -2907.713,E2 -2907.713} C_VEL
LIN {X 0,Y 559.15,Z 265.144,A -85,B 0,C 180,E1 -2910.183,E2 -2910.183} C_VEL
LIN {X 0,Y 559.171,Z 265.149,A -85,B 0,C 180,E1 -2912.714,E2 -2912.714} C_VEL
LIN {X 0,Y 559.155,Z 265.144,A -85,B 0,C 180,E1 -2915.322,E2 -2915.322} C_VEL
LIN {X 0,Y 559.13,Z 265.146,A -85,B 0,C 180,E1 -2918.018,E2 -2918.018} C_VEL
LIN {X 0,Y 559.174,Z 265.149,A -85,B 0,C 180,E1 -2920.811,E2 -2920.811} C_VEL
LIN {X 0,Y 559.138,Z 265.145,A -85,B 0,C 180,E1 -2923.734,E2 -2923.734} C_VEL
LIN {X 0,Y 559.165,Z 265.15,A -85,B 0,C 180,E1 -2926.801,E2 -2926.801} C_VEL
LIN {X 0,Y 559.174,Z 265.143,A -85,B 0,C 180,E1 -2929.19,E2 -2929.19} C_VEL
LIN {X 0,Y 559.13,Z 265.146,A -85,B 0,C 180,E1 -2931.983,E2 -2931.983} C_VEL
LIN {X 0,Y 559.129,Z 265.149,A -85,B 0,C 180,E1 -2934.787,E2 -2934.787} C_VEL
LIN {X 0,Y 559.153,Z 265.144,A -85,B 0,C 180,E1 -2937.365,E2 -2937.365} C_VEL
LIN {X 0,Y 559.146,Z 265.148,A -85,B 0,C 180,E1 -2940.143,E2 -2940.143} C_VEL
LIN {X 0,Y 559.179,Z 265.225,A -85,B 0,C 180,E1 -2941.407,E2 -2941.407} C_VEL
LIN {X 0,Y 562.249,Z 276.122,A -85,B 0,C 180,E1 -2942.559,E2 -2942.559} C_VEL
LIN {X 0,Y 561.755,Z 303.93,A -85,B 0,C 180,E1 -2945.024,E2 -2945.024} C_VEL
LIN {X 0,Y 561.671,Z 312.395,A -85,B 0,C 180,E1 -2945.743,E2 -2945.743} C_VEL
LIN {X 0,Y 563.181,Z 320.29,A -85,B 0,C 180,E1 -2945.92,E2 -2945.92} C_VEL
LIN {X 0,Y 562.284,Z 517.948,A -85,B 0,C 180,E1 -2948.58,E2 -2948.58} C_VEL
LIN {X 0,Y 562.07,Z 534.183,A -85,B 0,C 180,E1 -2948.932,E2 -2948.932} C_VEL
LIN {X 0,Y 561.787,Z 550.944,A -85,B 0,C 180,E1 -2949.448,E2 -2949.448} C_VEL
LIN {X 0,Y 561.511,Z 565.852,A -85,B 0,C 180,E1 -2950.046,E2 -2950.046} C_VEL
LIN {X 0,Y 561.137,Z 581.037,A -85,B 0,C 180,E1 -2950.806,E2 -2950.806} C_VEL
LIN {X 0,Y 560.779,Z 594.851,A -85,B 0,C 180,E1 -2951.647,E2 -2951.647} C_VEL
LIN {X 0,Y 560.367,Z 609.045,A -85,B 0,C 180,E1 -2952.671,E2 -2952.671} C_VEL
LIN {X 0,Y 559.988,Z 622.119,A -85,B 0,C 180,E1 -2953.785,E2 -2953.785} C_VEL
LIN {X 0,Y 559.722,Z 634.656,A -85,B 0,C 180,E1 -2955.044,E2 -2955.044} C_VEL
LIN {X 0,Y 559.448,Z 645.907,A -85,B 0,C 180,E1 -2956.376,E2 -2956.376} C_VEL
LIN {X 0,Y 559.219,Z 656.442,A -85,B 0,C 180,E1 -2957.848,E2 -2957.848} C_VEL
LIN {X 0,Y 559.057,Z 665.277,A -85,B 0,C 180,E1 -2959.314,E2 -2959.314} C_VEL
LIN {X 0,Y 558.93,Z 671.857,A -85,B 0,C 180,E1 -2960.592,E2 -2960.592} C_VEL
LIN {X 0,Y 558.893,Z 679.466,A -85,B 0,C 180,E1 -2962.413,E2 -2962.413} C_VEL
LIN {X 0,Y 558.863,Z 685.248,A -85,B 0,C 180,E1 -2964.226,E2 -2964.226} C_VEL
LIN {X 0,Y 558.805,Z 688.636,A -85,B 0,C 180,E1 -2965.672,E2 -2965.672} C_VEL
LIN {X 0,Y 558.787,Z 691.09,A -85,B 0,C 180,E1 -2967.116,E2 -2967.116} C_VEL
LIN {X 0,Y 558.739,Z 692.48,A -85,B 0,C 180,E1 -2968.559,E2 -2968.559} C_VEL
LIN {X 0,Y 558.735,Z 693,A -85,B 0,C 180,E1 -2970,E2 -2970} C_VEL
LIN {X 0,Y 558.738,Z 692.479,A -85,B 0,C 180,E1 -2971.442,E2 -2971.442} C_VEL
LIN {X 0,Y 558.787,Z 691.089,A -85,B 0,C 180,E1 -2972.884,E2 -2972.884} C_VEL
LIN {X 0,Y 558.805,Z 688.636,A -85,B 0,C 180,E1 -2974.328,E2 -2974.328} C_VEL
LIN {X 0,Y 558.862,Z 685.25,A -85,B 0,C 180,E1 -2975.774,E2 -2975.774} C_VEL
LIN {X 0,Y 558.893,Z 679.468,A -85,B 0,C 180,E1 -2977.587,E2 -2977.587} C_VEL
LIN {X 0,Y 558.93,Z 671.857,A -85,B 0,C 180,E1 -2979.408,E2 -2979.408} C_VEL
LIN {X 0,Y 559.116,Z 663.281,A -85,B 0,C 180,E1 -2981.046,E2 -2981.046} C_VEL
LIN {X 0,Y 559.275,Z 653.976,A -85,B 0,C 180,E1 -2982.519,E2 -2982.519} C_VEL
LIN {X 0,Y 559.471,Z 644.423,A -85,B 0,C 180,E1 -2983.808,E2 -2983.808} C_VEL
LIN {X 0,Y 559.791,Z 633.26,A -85,B 0,C 180,E1 -2985.103,E2 -2985.103} C_VEL
LIN {X 0,Y 560.05,Z 621.141,A -85,B 0,C 180,E1 -2986.307,E2 -2986.307} C_VEL
LIN {X 0,Y 560.419,Z 607.871,A -85,B 0,C 180,E1 -2987.422,E2 -2987.422} C_VEL
LIN {X 0,Y 560.807,Z 593.422,A -85,B 0,C 180,E1 -2988.447,E2 -2988.447} C_VEL
LIN {X 0,Y 561.19,Z 579.278,A -85,B 0,C 180,E1 -2989.287,E2 -2989.287} C_VEL
LIN {X 0,Y 561.546,Z 564.537,A -85,B 0,C 180,E1 -2990.014,E2 -2990.014} C_VEL
LIN {X 0,Y 561.868,Z 548.345,A -85,B 0,C 180,E1 -2990.645,E2 -2990.645} C_VEL
LIN {X 0,Y 562.134,Z 532.354,A -85,B 0,C 180,E1 -2991.114,E2 -2991.114} C_VEL
LIN {X 0,Y 562.29,Z 516.441,A -85,B 0,C 180,E1 -2991.444,E2 -2991.444} C_VEL
LIN {X 0,Y 563.201,Z 321.006,A -85,B 0,C 180,E1 -2994.069,E2 -2994.069} C_VEL
LIN {X 0,Y 561.62,Z 311.979,A -85,B 0,C 180,E1 -2994.27,E2 -2994.27} C_VEL
LIN {X 0,Y 562.281,Z 278.301,A -85,B 0,C 180,E1 -2997.243,E2 -2997.243} C_VEL
LIN {X 0,Y 562.05,Z 274.941,A -85,B 0,C 180,E1 -2997.558,E2 -2997.558} C_VEL
LIN {X 0,Y 559.175,Z 265.145,A -85,B 0,C 180,E1 -2998.606,E2 -2998.606} C_VEL
LIN {X 0,Y 559.147,Z 265.152,A -85,B 0,C 180,E1 -3001.274,E2 -3001.274} C_VEL
LIN {X 0,Y 559.163,Z 265.143,A -85,B 0,C 180,E1 -3003.949,E2 -3003.949} C_VEL
LIN {X 0,Y 559.139,Z 265.151,A -85,B 0,C 180,E1 -3007.108,E2 -3007.108} C_VEL
LIN {X 0,Y 559.162,Z 265.143,A -85,B 0,C 180,E1 -3009.942,E2 -3009.942} C_VEL
LIN {X 0,Y 559.161,Z 265.143,A -85,B 0,C 180,E1 -3012.743,E2 -3012.743} C_VEL
LIN {X 0,Y 559.15,Z 265.143,A -85,B 0,C 180,E1 -3015.761,E2 -3015.761} C_VEL
LIN {X 0,Y 559.189,Z 265.136,A -85,B 0,C 180,E1 -3018.232,E2 -3018.232} C_VEL
LIN {X 0,Y 559.172,Z 265.147,A -85,B 0,C 180,E1 -3021.192,E2 -3021.192} C_VEL
LIN {X 0,Y 559.159,Z 265.142,A -85,B 0,C 180,E1 -3023.791,E2 -3023.791} C_VEL
LIN {X 0,Y 559.16,Z 265.141,A -85,B 0,C 180,E1 -3026.425,E2 -3026.425} C_VEL
LIN {X 0,Y 559.153,Z 265.148,A -85,B 0,C 180,E1 -3028.981,E2 -3028.981} C_VEL
LIN {X 0,Y 559.165,Z 265.143,A -85,B 0,C 180,E1 -3031.619,E2 -3031.619} C_VEL
LIN {X 0,Y 559.177,Z 265.139,A -85,B 0,C 180,E1 -3033.903,E2 -3033.903} C_VEL
LIN {X 0,Y 559.154,Z 265.143,A -85,B 0,C 180,E1 -3036.567,E2 -3036.567} C_VEL
LIN {X 0,Y 559.174,Z 265.139,A -85,B 0,C 180,E1 -3039.395,E2 -3039.395} C_VEL
LIN {X 0,Y 559.141,Z 265.145,A -85,B 0,C 180,E1 -3041.686,E2 -3041.686} C_VEL
LIN {X 0,Y 559.164,Z 265.14,A -85,B 0,C 180,E1 -3043.948,E2 -3043.948} C_VEL
LIN {X 0,Y 559.169,Z 265.135,A -85,B 0,C 180,E1 -3046.184,E2 -3046.184} C_VEL
LIN {X 0,Y 559.193,Z 265.146,A -85,B 0,C 180,E1 -3049.134,E2 -3049.134} C_VEL
LIN {X 0,Y 559.201,Z 265.133,A -85,B 0,C 180,E1 -3052.054,E2 -3052.054} C_VEL
LIN {X 0,Y 559.252,Z 265.132,A -85,B 0,C 180,E1 -3054.953,E2 -3054.953} C_VEL
LIN {X 0,Y 559.254,Z 265.129,A -85,B 0,C 180,E1 -3057.84,E2 -3057.84} C_VEL
LIN {X 0,Y 559.269,Z 265.128,A -85,B 0,C 180,E1 -3060.72,E2 -3060.72} C_VEL
LIN {X 0,Y 559.236,Z 265.136,A -85,B 0,C 180,E1 -3062.881,E2 -3062.881} C_VEL
LIN {X 0,Y 559.23,Z 265.131,A -85,B 0,C 180,E1 -3065.77,E2 -3065.77} C_VEL
LIN {X 0,Y 559.185,Z 265.136,A -85,B 0,C 180,E1 -3068.675,E2 -3068.675} C_VEL
LIN {X 0,Y 559.203,Z 265.137,A -85,B 0,C 180,E1 -3071.601,E2 -3071.601} C_VEL
LIN {X 0,Y 559.198,Z 265.137,A -85,B 0,C 180,E1 -3074.596,E2 -3074.596} C_VEL
LIN {X 0,Y 559.157,Z 265.143,A -85,B 0,C 180,E1 -3077.557,E2 -3077.557} C_VEL
LIN {X 0,Y 559.17,Z 265.139,A -85,B 0,C 180,E1 -3079.838,E2 -3079.838} C_VEL
LIN {X 0,Y 559.139,Z 265.138,A -85,B 0,C 180,E1 -3082.153,E2 -3082.153} C_VEL
LIN {X 0,Y 559.177,Z 265.144,A -85,B 0,C 180,E1 -3085.187,E2 -3085.187} C_VEL
LIN {X 0,Y 559.155,Z 265.137,A -85,B 0,C 180,E1 -3087.714,E2 -3087.714} C_VEL
LIN {X 0,Y 559.138,Z 265.146,A -85,B 0,C 180,E1 -3090.612,E2 -3090.612} C_VEL
LIN {X 0,Y 558.476,Z 265.233,A -85,B 0,C 180,E1 -3091.214,E2 -3091.214} C_VEL
LIN {X 0,Y 555.613,Z 265.588,A -85,B 0,C 180,E1 -3092.19,E2 -3092.19} C_VEL
LIN {X 0,Y 553.202,Z 265.891,A -85,B 0,C 180,E1 -3092.975,E2 -3092.975} C_VEL
LIN {X 0,Y 552.184,Z 266.011,A -85,B 0,C 180,E1 -3093.582,E2 -3093.582} C_VEL
LIN {X 0,Y 552.111,Z 266.019,A -85,B 0,C 180,E1 -3093.787,E2 -3093.787} C_VEL
LIN {X 0,Y 552.111,Z 266.027,A -85,B 0,C 180,E1 -3096.747,E2 -3096.747} C_VEL
LIN {X 0,Y 552.129,Z 266.017,A -85,B 0,C 180,E1 -3099.527,E2 -3099.527} C_VEL
LIN {X 0,Y 552.129,Z 266.017,A -85,B 0,C 180,E1 -3102.426,E2 -3102.426} C_VEL
LIN {X 0,Y 552.099,Z 266.018,A -85,B 0,C 180,E1 -3105.563,E2 -3105.563} C_VEL
LIN {X 0,Y 552.14,Z 266.024,A -85,B 0,C 180,E1 -3108.676,E2 -3108.676} C_VEL
LIN {X 0,Y 552.119,Z 266.018,A -85,B 0,C 180,E1 -3111.411,E2 -3111.411} C_VEL
LIN {X 0,Y 552.084,Z 266.022,A -85,B 0,C 180,E1 -3114.157,E2 -3114.157} C_VEL
LIN {X 0,Y 552.115,Z 266.021,A -85,B 0,C 180,E1 -3116.814,E2 -3116.814} C_VEL
LIN {X 0,Y 552.104,Z 266.024,A -85,B 0,C 180,E1 -3119.391,E2 -3119.391} C_VEL
LIN {X 0,Y 552.106,Z 266.024,A -85,B 0,C 180,E1 -3121.902,E2 -3121.902} C_VEL
LIN {X 0,Y 552.134,Z 266.051,A -85,B 0,C 180,E1 -3123.544,E2 -3123.544} C_VEL
LIN {X 0,Y 554.673,Z 275.604,A -85,B 0,C 180,E1 -3124.683,E2 -3124.683} C_VEL
LIN {X 0,Y 554.702,Z 283.117,A -85,B 0,C 180,E1 -3125.464,E2 -3125.464} C_VEL
LIN {X 0,Y 556.741,Z 293.403,A -85,B 0,C 180,E1 -3125.708,E2 -3125.708} C_VEL
LIN {X 0,Y 555.659,Z 488.177,A -85,B 0,C 180,E1 -3128.36,E2 -3128.36} C_VEL
LIN {X 0,Y 555.435,Z 504.322,A -85,B 0,C 180,E1 -3128.716,E2 -3128.716} C_VEL
LIN {X 0,Y 555.128,Z 521.036,A -85,B 0,C 180,E1 -3129.238,E2 -3129.238} C_VEL
LIN {X 0,Y 554.787,Z 536.393,A -85,B 0,C 180,E1 -3129.865,E2 -3129.865} C_VEL
LIN {X 0,Y 554.372,Z 551.954,A -85,B 0,C 180,E1 -3130.659,E2 -3130.659} C_VEL
LIN {X 0,Y 553.92,Z 567.166,A -85,B 0,C 180,E1 -3131.612,E2 -3131.612} C_VEL
LIN {X 0,Y 553.466,Z 580.955,A -85,B 0,C 180,E1 -3132.648,E2 -3132.648} C_VEL
LIN {X 0,Y 553.072,Z 593.603,A -85,B 0,C 180,E1 -3133.766,E2 -3133.766} C_VEL
LIN {X 0,Y 552.738,Z 604.896,A -85,B 0,C 180,E1 -3134.923,E2 -3134.923} C_VEL
LIN {X 0,Y 552.449,Z 615.551,A -85,B 0,C 180,E1 -3136.2,E2 -3136.2} C_VEL
LIN {X 0,Y 552.227,Z 624.913,A -85,B 0,C 180,E1 -3137.505,E2 -3137.505} C_VEL
LIN {X 0,Y 552.04,Z 634.022,A -85,B 0,C 180,E1 -3138.991,E2 -3138.991} C_VEL
LIN {X 0,Y 551.87,Z 641.638,A -85,B 0,C 180,E1 -3140.471,E2 -3140.471} C_VEL
LIN {X 0,Y 551.83,Z 647.876,A -85,B 0,C 180,E1 -3141.947,E2 -3141.947} C_VEL
LIN {X 0,Y 551.763,Z 653.147,A -85,B 0,C 180,E1 -3143.471,E2 -3143.471} C_VEL
LIN {X 0,Y 551.697,Z 656.952,A -85,B 0,C 180,E1 -3144.884,E2 -3144.884} C_VEL
LIN {X 0,Y 551.729,Z 659.909,A -85,B 0,C 180,E1 -3146.348,E2 -3146.348} C_VEL
LIN {X 0,Y 551.652,Z 661.846,A -85,B 0,C 180,E1 -3147.81,E2 -3147.81} C_VEL
LIN {X 0,Y 551.637,Z 662.839,A -85,B 0,C 180,E1 -3149.27,E2 -3149.27} C_VEL
LIN {X 0,Y 551.636,Z 662.858,A -85,B 0,C 180,E1 -3150.73,E2 -3150.73} C_VEL
LIN {X 0,Y 551.652,Z 661.943,A -85,B 0,C 180,E1 -3152.19,E2 -3152.19} C_VEL
LIN {X 0,Y 551.728,Z 660.049,A -85,B 0,C 180,E1 -3153.652,E2 -3153.652} C_VEL
LIN {X 0,Y 551.695,Z 657.17,A -85,B 0,C 180,E1 -3155.116,E2 -3155.116} C_VEL
LIN {X 0,Y 551.763,Z 653.252,A -85,B 0,C 180,E1 -3156.583,E2 -3156.583} C_VEL
LIN {X 0,Y 551.825,Z 648.222,A -85,B 0,C 180,E1 -3158.053,E2 -3158.053} C_VEL
LIN {X 0,Y 551.858,Z 642.066,A -85,B 0,C 180,E1 -3159.529,E2 -3159.529} C_VEL
LIN {X 0,Y 552.097,Z 633.049,A -85,B 0,C 180,E1 -3161.276,E2 -3161.276} C_VEL
LIN {X 0,Y 552.256,Z 624.275,A -85,B 0,C 180,E1 -3162.681,E2 -3162.681} C_VEL
LIN {X 0,Y 552.48,Z 614.778,A -85,B 0,C 180,E1 -3163.986,E2 -3163.986} C_VEL
LIN {X 0,Y 552.819,Z 603.711,A -85,B 0,C 180,E1 -3165.295,E2 -3165.295} C_VEL
LIN {X 0,Y 553.179,Z 590.61,A -85,B 0,C 180,E1 -3166.61,E2 -3166.61} C_VEL
LIN {X 0,Y 553.598,Z 577.248,A -85,B 0,C 180,E1 -3167.739,E2 -3167.739} C_VEL
LIN {X 0,Y 553.987,Z 564.09,A -85,B 0,C 180,E1 -3168.682,E2 -3168.682} C_VEL
LIN {X 0,Y 554.447,Z 548.339,A -85,B 0,C 180,E1 -3169.627,E2 -3169.627} C_VEL
LIN {X 0,Y 554.821,Z 532.832,A -85,B 0,C 180,E1 -3170.386,E2 -3170.386} C_VEL
LIN {X 0,Y 555.269,Z 516.908,A -85,B 0,C 180,E1 -3170.999,E2 -3170.999} C_VEL
LIN {X 0,Y 555.526,Z 500.381,A -85,B 0,C 180,E1 -3171.474,E2 -3171.474} C_VEL
LIN {X 0,Y 555.695,Z 484.706,A -85,B 0,C 180,E1 -3171.784,E2 -3171.784} C_VEL
LIN {X 0,Y 556.69,Z 292.959,A -85,B 0,C 180,E1 -3174.39,E2 -3174.39} C_VEL
LIN {X 0,Y 554.689,Z 283.083,A -85,B 0,C 180,E1 -3174.63,E2 -3174.63} C_VEL
LIN {X 0,Y 554.8,Z 276.483,A -85,B 0,C 180,E1 -3175.311,E2 -3175.311} C_VEL
LIN {X 0,Y 552.121,Z 266.025,A -85,B 0,C 180,E1 -3176.58,E2 -3176.58} C_VEL
LIN {X 0,Y 552.109,Z 266.023,A -85,B 0,C 180,E1 -3179.765,E2 -3179.765} C_VEL
LIN {X 0,Y 552.114,Z 266.02,A -85,B 0,C 180,E1 -3182.318,E2 -3182.318} C_VEL
LIN {X 0,Y 552.081,Z 266.03,A -85,B 0,C 180,E1 -3184.949,E2 -3184.949} C_VEL
LIN {X 0,Y 552.092,Z 266.024,A -85,B 0,C 180,E1 -3187.885,E2 -3187.885} C_VEL
LIN {X 0,Y 552.108,Z 266.02,A -85,B 0,C 180,E1 -3190.481,E2 -3190.481} C_VEL
LIN {X 0,Y 552.113,Z 266.025,A -85,B 0,C 180,E1 -3193.484,E2 -3193.484} C_VEL
LIN {X 0,Y 552.105,Z 266.02,A -85,B 0,C 180,E1 -3196.576,E2 -3196.576} C_VEL
LIN {X 0,Y 552.108,Z 266.024,A -85,B 0,C 180,E1 -3199.519,E2 -3199.519} C_VEL
LIN {X 0,Y 552.091,Z 266.02,A -85,B 0,C 180,E1 -3202.336,E2 -3202.336} C_VEL
LIN {X 0,Y 552.119,Z 266.025,A -85,B 0,C 180,E1 -3205.053,E2 -3205.053} C_VEL
LIN {X 0,Y 552.113,Z 266.019,A -85,B 0,C 180,E1 -3207.681,E2 -3207.681} C_VEL
LIN {X 0,Y 552.109,Z 266.019,A -85,B 0,C 180,E1 -3210.235,E2 -3210.235} C_VEL
LIN {X 0,Y 552.136,Z 266.019,A -85,B 0,C 180,E1 -3213,E2 -3213} C_VEL
LIN {X 0,Y 552.112,Z 266.028,A -85,B 0,C 180,E1 -3215.161,E2 -3215.161} C_VEL
LIN {X 0,Y 552.093,Z 266.02,A -85,B 0,C 180,E1 -3217.549,E2 -3217.549} C_VEL
LIN {X 0,Y 552.141,Z 266.016,A -85,B 0,C 180,E1 -3220.375,E2 -3220.375} C_VEL
LIN {X 0,Y 552.153,Z 266.02,A -85,B 0,C 180,E1 -3222.977,E2 -3222.977} C_VEL
LIN {X 0,Y 552.133,Z 266.016,A -85,B 0,C 180,E1 -3226.004,E2 -3226.004} C_VEL
LIN {X 0,Y 552.16,Z 266.019,A -85,B 0,C 180,E1 -3228.993,E2 -3228.993} C_VEL
LIN {X 0,Y 552.155,Z 266.012,A -85,B 0,C 180,E1 -3231.951,E2 -3231.951} C_VEL
LIN {X 0,Y 552.227,Z 266.012,A -85,B 0,C 180,E1 -3234.889,E2 -3234.889} C_VEL
LIN {X 0,Y 552.224,Z 266.001,A -85,B 0,C 180,E1 -3237.812,E2 -3237.812} C_VEL
LIN {X 0,Y 552.24,Z 266.008,A -85,B 0,C 180,E1 -3240.729,E2 -3240.729} C_VEL
LIN {X 0,Y 552.202,Z 266.013,A -85,B 0,C 180,E1 -3242.918,E2 -3242.918} C_VEL
LIN {X 0,Y 552.205,Z 266.006,A -85,B 0,C 180,E1 -3245.844,E2 -3245.844} C_VEL
LIN {X 0,Y 552.155,Z 266.02,A -85,B 0,C 180,E1 -3248.786,E2 -3248.786} C_VEL
LIN {X 0,Y 552.16,Z 266.011,A -85,B 0,C 180,E1 -3251.75,E2 -3251.75} C_VEL
LIN {X 0,Y 552.134,Z 266.023,A -85,B 0,C 180,E1 -3254.748,E2 -3254.748} C_VEL
LIN {X 0,Y 552.108,Z 266.019,A -85,B 0,C 180,E1 -3257.788,E2 -3257.788} C_VEL
LIN {X 0,Y 552.128,Z 266.018,A -85,B 0,C 180,E1 -3260.101,E2 -3260.101} C_VEL
LIN {X 0,Y 552.093,Z 266.025,A -85,B 0,C 180,E1 -3262.451,E2 -3262.451} C_VEL
LIN {X 0,Y 552.152,Z 266.017,A -85,B 0,C 180,E1 -3265.35,E2 -3265.35} C_VEL
LIN {X 0,Y 552.106,Z 266.021,A -85,B 0,C 180,E1 -3268.098,E2 -3268.098} C_VEL
LIN {X 0,Y 552.1,Z 266.027,A -85,B 0,C 180,E1 -3270.609,E2 -3270.609} C_VEL
LIN {X 0,Y 552.12,Z 266.023,A -85,B 0,C 180,E1 -3273.185,E2 -3273.185} C_VEL
LIN {X 0,Y 552.111,Z 266.019,A -85,B 0,C 180,E1 -3275.842,E2 -3275.842} C_VEL
LIN {X 0,Y 552.119,Z 266.025,A -85,B 0,C 180,E1 -3279.061,E2 -3279.061} C_VEL
LIN {X 0,Y 552.137,Z 266.018,A -85,B 0,C 180,E1 -3281.444,E2 -3281.444} C_VEL
LIN {X 0,Y 552.092,Z 266.029,A -85,B 0,C 180,E1 -3284.532,E2 -3284.532} C_VEL
LIN {X 0,Y 552.128,Z 266.018,A -85,B 0,C 180,E1 -3287.585,E2 -3287.585} C_VEL
LIN {X 0,Y 552.128,Z 266.024,A -85,B 0,C 180,E1 -3290.473,E2 -3290.473} C_VEL
LIN {X 0,Y 552.104,Z 266.023,A -85,B 0,C 180,E1 -3293.317,E2 -3293.317} C_VEL
LIN {X 0,Y 552.124,Z 266.015,A -85,B 0,C 180,E1 -3295.939,E2 -3295.939} C_VEL
LIN {X 0,Y 552.117,Z 266.027,A -85,B 0,C 180,E1 -3298.541,E2 -3298.541} C_VEL
LIN {X 0,Y 552.128,Z 266.143,A -85,B 0,C 180,E1 -3301.113,E2 -3301.113} C_VEL
LIN {X 0,Y 555.632,Z 278.415,A -85,B 0,C 180,E1 -3302.432,E2 -3302.432} C_VEL
LIN {X 0,Y 554.961,Z 308.186,A -85,B 0,C 180,E1 -3305.098,E2 -3305.098} C_VEL
LIN {X 0,Y 554.89,Z 311.779,A -85,B 0,C 180,E1 -3305.417,E2 -3305.417} C_VEL
LIN {X 0,Y 556.735,Z 322.378,A -85,B 0,C 180,E1 -3305.654,E2 -3305.654} C_VEL
LIN {X 0,Y 555.667,Z 519.438,A -85,B 0,C 180,E1 -3308.336,E2 -3308.336} C_VEL
LIN {X 0,Y 555.443,Z 536.014,A -85,B 0,C 180,E1 -3308.717,E2 -3308.717} C_VEL
LIN {X 0,Y 555.086,Z 552.243,A -85,B 0,C 180,E1 -3309.237,E2 -3309.237} C_VEL
LIN {X 0,Y 554.724,Z 568.735,A -85,B 0,C 180,E1 -3309.931,E2 -3309.931} C_VEL
LIN {X 0,Y 554.34,Z 582.712,A -85,B 0,C 180,E1 -3310.658,E2 -3310.658} C_VEL
LIN {X 0,Y 553.933,Z 597.69,A -85,B 0,C 180,E1 -3311.603,E2 -3311.603} C_VEL
LIN {X 0,Y 553.461,Z 611.605,A -85,B 0,C 180,E1 -3312.656,E2 -3312.656} C_VEL
LIN {X 0,Y 553.046,Z 624.068,A -85,B 0,C 180,E1 -3313.766,E2 -3313.766} C_VEL
LIN {X 0,Y 552.786,Z 634.979,A -85,B 0,C 180,E1 -3314.889,E2 -3314.889} C_VEL
LIN {X 0,Y 552.445,Z 645.907,A -85,B 0,C 180,E1 -3316.2,E2 -3316.2} C_VEL
LIN {X 0,Y 552.209,Z 656.441,A -85,B 0,C 180,E1 -3317.691,E2 -3317.691} C_VEL
LIN {X 0,Y 551.992,Z 665.276,A -85,B 0,C 180,E1 -3319.176,E2 -3319.176} C_VEL
LIN {X 0,Y 551.861,Z 671.856,A -85,B 0,C 180,E1 -3320.471,E2 -3320.471} C_VEL
LIN {X 0,Y 551.804,Z 679.466,A -85,B 0,C 180,E1 -3322.315,E2 -3322.315} C_VEL
LIN {X 0,Y 551.77,Z 685.249,A -85,B 0,C 180,E1 -3324.152,E2 -3324.152} C_VEL
LIN {X 0,Y 551.702,Z 688.636,A -85,B 0,C 180,E1 -3325.617,E2 -3325.617} C_VEL
LIN {X 0,Y 551.711,Z 691.09,A -85,B 0,C 180,E1 -3327.079,E2 -3327.079} C_VEL
LIN {X 0,Y 551.638,Z 692.479,A -85,B 0,C 180,E1 -3328.54,E2 -3328.54} C_VEL
LIN {X 0,Y 551.636,Z 693,A -85,B 0,C 180,E1 -3330,E2 -3330} C_VEL
LIN {X 0,Y 551.638,Z 692.479,A -85,B 0,C 180,E1 -3331.46,E2 -3331.46} C_VEL
LIN {X 0,Y 551.711,Z 691.089,A -85,B 0,C 180,E1 -3332.921,E2 -3332.921} C_VEL
LIN {X 0,Y 551.702,Z 688.635,A -85,B 0,C 180,E1 -3334.384,E2 -3334.384} C_VEL
LIN {X 0,Y 551.77,Z 685.25,A -85,B 0,C 180,E1 -3335.848,E2 -3335.848} C_VEL
LIN {X 0,Y 551.804,Z 679.468,A -85,B 0,C 180,E1 -3337.685,E2 -3337.685} C_VEL
LIN {X 0,Y 551.86,Z 671.856,A -85,B 0,C 180,E1 -3339.53,E2 -3339.53} C_VEL
LIN {X 0,Y 552.04,Z 664.267,A -85,B 0,C 180,E1 -3341.009,E2 -3341.009} C_VEL
LIN {X 0,Y 552.226,Z 655.21,A -85,B 0,C 180,E1 -3342.495,E2 -3342.495} C_VEL
LIN {X 0,Y 552.483,Z 644.422,A -85,B 0,C 180,E1 -3343.986,E2 -3343.986} C_VEL
LIN {X 0,Y 552.855,Z 633.449,A -85,B 0,C 180,E1 -3345.277,E2 -3345.277} C_VEL
LIN {X 0,Y 553.161,Z 621.14,A -85,B 0,C 180,E1 -3346.516,E2 -3346.516} C_VEL
LIN {X 0,Y 553.578,Z 607.638,A -85,B 0,C 180,E1 -3347.663,E2 -3347.663} C_VEL
LIN {X 0,Y 553.987,Z 593.419,A -85,B 0,C 180,E1 -3348.683,E2 -3348.683} C_VEL
LIN {X 0,Y 554.413,Z 579.274,A -85,B 0,C 180,E1 -3349.532,E2 -3349.532} C_VEL
LIN {X 0,Y 554.846,Z 564.262,A -85,B 0,C 180,E1 -3350.278,E2 -3350.278} C_VEL
LIN {X 0,Y 555.217,Z 548.344,A -85,B 0,C 180,E1 -3350.904,E2 -3350.904} C_VEL
LIN {X 0,Y 555.502,Z 532.354,A -85,B 0,C 180,E1 -3351.378,E2 -3351.378} C_VEL
LIN {X 0,Y 555.683,Z 516.441,A -85,B 0,C 180,E1 -3351.712,E2 -3351.712} C_VEL
LIN {X 0,Y 556.723,Z 322.266,A -85,B 0,C 180,E1 -3354.348,E2 -3354.348} C_VEL
LIN {X 0,Y 554.918,Z 311.8,A -85,B 0,C 180,E1 -3354.58,E2 -3354.58} C_VEL
LIN {X 0,Y 555.637,Z 278.541,A -85,B 0,C 180,E1 -3357.556,E2 -3357.556} C_VEL
LIN {X 0,Y 552.117,Z 266.027,A -85,B 0,C 180,E1 -3358.928,E2 -3358.928} C_VEL
LIN {X 0,Y 552.109,Z 266.027,A -85,B 0,C 180,E1 -3361.475,E2 -3361.475} C_VEL
LIN {X 0,Y 552.13,Z 266.019,A -85,B 0,C 180,E1 -3364.17,E2 -3364.17} C_VEL
LIN {X 0,Y 552.103,Z 266.023,A -85,B 0,C 180,E1 -3366.747,E2 -3366.747} C_VEL
LIN {X 0,Y 552.13,Z 266.023,A -85,B 0,C 180,E1 -3369.527,E2 -3369.527} C_VEL
LIN {X 0,Y 552.129,Z 266.017,A -85,B 0,C 180,E1 -3372.425,E2 -3372.425} C_VEL
LIN {X 0,Y 552.095,Z 266.025,A -85,B 0,C 180,E1 -3375.563,E2 -3375.563} C_VEL
LIN {X 0,Y 552.138,Z 266.016,A -85,B 0,C 180,E1 -3378.676,E2 -3378.676} C_VEL
LIN {X 0,Y 552.115,Z 266.024,A -85,B 0,C 180,E1 -3381.411,E2 -3381.411} C_VEL
LIN {X 0,Y 552.101,Z 266.019,A -85,B 0,C 180,E1 -3384.158,E2 -3384.158} C_VEL
LIN {X 0,Y 552.112,Z 266.022,A -85,B 0,C 180,E1 -3386.814,E2 -3386.814} C_VEL
LIN {X 0,Y 552.1,Z 266.026,A -85,B 0,C 180,E1 -3389.391,E2 -3389.391} C_VEL
LIN {X 0,Y 552.106,Z 266.02,A -85,B 0,C 180,E1 -3391.902,E2 -3391.902} C_VEL
LIN {X 0,Y 552.153,Z 266.016,A -85,B 0,C 180,E1 -3394.65,E2 -3394.65} C_VEL
LIN {X 0,Y 552.093,Z 266.024,A -85,B 0,C 180,E1 -3397.549,E2 -3397.549} C_VEL
LIN {X 0,Y 552.141,Z 266.01,A -85,B 0,C 180,E1 -3400.375,E2 -3400.375} C_VEL
LIN {X 0,Y 552.153,Z 266.021,A -85,B 0,C 180,E1 -3402.977,E2 -3402.977} C_VEL
LIN {X 0,Y 552.133,Z 266.011,A -85,B 0,C 180,E1 -3406.005,E2 -3406.005} C_VEL
LIN {X 0,Y 552.16,Z 266.019,A -85,B 0,C 180,E1 -3408.993,E2 -3408.993} C_VEL
LIN {X 0,Y 552.155,Z 266.011,A -85,B 0,C 180,E1 -3411.952,E2 -3411.952} C_VEL
LIN {X 0,Y 552.228,Z 266.006,A -85,B 0,C 180,E1 -3414.889,E2 -3414.889} C_VEL
LIN {X 0,Y 552.225,Z 266.005,A -85,B 0,C 180,E1 -3417.812,E2 -3417.812} C_VEL
LIN {X 0,Y 552.239,Z 266.003,A -85,B 0,C 180,E1 -3420.729,E2 -3420.729} C_VEL
LIN {X 0,Y 552.202,Z 266.012,A -85,B 0,C 180,E1 -3422.918,E2 -3422.918} C_VEL
LIN {X 0,Y 552.199,Z 266.007,A -85,B 0,C 180,E1 -3425.844,E2 -3425.844} C_VEL
LIN {X 0,Y 552.156,Z 266.012,A -85,B 0,C 180,E1 -3428.786,E2 -3428.786} C_VEL
LIN {X 0,Y 552.161,Z 266.013,A -85,B 0,C 180,E1 -3431.751,E2 -3431.751} C_VEL
LIN {X 0,Y 552.135,Z 266.019,A -85,B 0,C 180,E1 -3434.749,E2 -3434.749} C_VEL
LIN {X 0,Y 552.108,Z 266.019,A -85,B 0,C 180,E1 -3437.789,E2 -3437.789} C_VEL
LIN {X 0,Y 552.129,Z 266.016,A -85,B 0,C 180,E1 -3440.101,E2 -3440.101} C_VEL
LIN {X 0,Y 552.094,Z 266.017,A -85,B 0,C 180,E1 -3442.451,E2 -3442.451} C_VEL
LIN {X 0,Y 552.153,Z 266.016,A -85,B 0,C 180,E1 -3445.351,E2 -3445.351} C_VEL
LIN {X 0,Y 552.107,Z 266.014,A -85,B 0,C 180,E1 -3448.099,E2 -3448.099} C_VEL
LIN {X 0,Y 552.101,Z 266.025,A -85,B 0,C 180,E1 -3450.609,E2 -3450.609} C_VEL
LIN {X 0,Y 552.114,Z 266.023,A -85,B 0,C 180,E1 -3453.186,E2 -3453.186} C_VEL
LIN {X 0,Y 552.111,Z 266.019,A -85,B 0,C 180,E1 -3453.787,E2 -3453.787} C_VEL
LIN {X 0,Y 551.48,Z 266.101,A -85,B 0,C 180,E1 -3454.396,E2 -3454.396} C_VEL
LIN {X 0,Y 548.66,Z 266.457,A -85,B 0,C 180,E1 -3455.384,E2 -3455.384} C_VEL
LIN {X 0,Y 546.239,Z 266.761,A -85,B 0,C 180,E1 -3456.18,E2 -3456.18} C_VEL
LIN {X 0,Y 545.168,Z 266.891,A -85,B 0,C 180,E1 -3456.794,E2 -3456.794} C_VEL
LIN {X 0,Y 545.065,Z 266.9,A -85,B 0,C 180,E1 -3457.002,E2 -3457.002} C_VEL
LIN {X 0,Y 545.065,Z 266.897,A -85,B 0,C 180,E1 -3460.143,E2 -3460.143} C_VEL
LIN {X 0,Y 545.077,Z 266.901,A -85,B 0,C 180,E1 -3463.107,E2 -3463.107} C_VEL
LIN {X 0,Y 545.058,Z 266.896,A -85,B 0,C 180,E1 -3466.225,E2 -3466.225} C_VEL
LIN {X 0,Y 545.096,Z 266.902,A -85,B 0,C 180,E1 -3468.887,E2 -3468.887} C_VEL
LIN {X 0,Y 545.053,Z 266.896,A -85,B 0,C 180,E1 -3471.763,E2 -3471.763} C_VEL
LIN {X 0,Y 545.035,Z 266.905,A -85,B 0,C 180,E1 -3474.532,E2 -3474.532} C_VEL
LIN {X 0,Y 545.068,Z 266.899,A -85,B 0,C 180,E1 -3477.212,E2 -3477.212} C_VEL
LIN {X 0,Y 545.064,Z 266.9,A -85,B 0,C 180,E1 -3479.811,E2 -3479.811} C_VEL
LIN {X 0,Y 545.093,Z 266.903,A -85,B 0,C 180,E1 -3482.827,E2 -3482.827} C_VEL
LIN {X 0,Y 545.118,Z 266.996,A -85,B 0,C 180,E1 -3483.255,E2 -3483.255} C_VEL
LIN {X 0,Y 548.056,Z 277.973,A -85,B 0,C 180,E1 -3484.583,E2 -3484.583} C_VEL
LIN {X 0,Y 548.043,Z 283.329,A -85,B 0,C 180,E1 -3485.146,E2 -3485.146} C_VEL
LIN {X 0,Y 550.254,Z 294.185,A -85,B 0,C 180,E1 -3485.411,E2 -3485.411} C_VEL
LIN {X 0,Y 549.081,Z 486.878,A -85,B 0,C 180,E1 -3488.063,E2 -3488.063} C_VEL
LIN {X 0,Y 548.859,Z 503.567,A -85,B 0,C 180,E1 -3488.424,E2 -3488.424} C_VEL
LIN {X 0,Y 548.526,Z 519.849,A -85,B 0,C 180,E1 -3488.928,E2 -3488.928} C_VEL
LIN {X 0,Y 548.126,Z 535.23,A -85,B 0,C 180,E1 -3489.55,E2 -3489.55} C_VEL
LIN {X 0,Y 547.65,Z 550.221,A -85,B 0,C 180,E1 -3490.314,E2 -3490.314} C_VEL
LIN {X 0,Y 547.22,Z 564.18,A -85,B 0,C 180,E1 -3491.175,E2 -3491.175} C_VEL
LIN {X 0,Y 546.732,Z 577.765,A -85,B 0,C 180,E1 -3492.164,E2 -3492.164} C_VEL
LIN {X 0,Y 546.271,Z 590.67,A -85,B 0,C 180,E1 -3493.27,E2 -3493.27} C_VEL
LIN {X 0,Y 545.909,Z 602.867,A -85,B 0,C 180,E1 -3494.506,E2 -3494.506} C_VEL
LIN {X 0,Y 545.524,Z 614.07,A -85,B 0,C 180,E1 -3495.831,E2 -3495.831} C_VEL
LIN {X 0,Y 545.21,Z 624.916,A -85,B 0,C 180,E1 -3497.342,E2 -3497.342} C_VEL
LIN {X 0,Y 545.016,Z 634.026,A -85,B 0,C 180,E1 -3498.847,E2 -3498.847} C_VEL
LIN {X 0,Y 544.803,Z 641.64,A -85,B 0,C 180,E1 -3500.346,E2 -3500.346} C_VEL
LIN {X 0,Y 544.743,Z 647.878,A -85,B 0,C 180,E1 -3501.841,E2 -3501.841} C_VEL
LIN {X 0,Y 544.679,Z 653.419,A -85,B 0,C 180,E1 -3503.48,E2 -3503.48} C_VEL
LIN {X 0,Y 544.62,Z 656.953,A -85,B 0,C 180,E1 -3504.817,E2 -3504.817} C_VEL
LIN {X 0,Y 544.643,Z 659.91,A -85,B 0,C 180,E1 -3506.301,E2 -3506.301} C_VEL
LIN {X 0,Y 544.566,Z 661.847,A -85,B 0,C 180,E1 -3507.781,E2 -3507.781} C_VEL
LIN {X 0,Y 544.537,Z 662.838,A -85,B 0,C 180,E1 -3509.26,E2 -3509.26} C_VEL
LIN {X 0,Y 544.537,Z 662.858,A -85,B 0,C 180,E1 -3510.739,E2 -3510.739} C_VEL
LIN {X 0,Y 544.567,Z 661.943,A -85,B 0,C 180,E1 -3512.219,E2 -3512.219} C_VEL
LIN {X 0,Y 544.643,Z 660.047,A -85,B 0,C 180,E1 -3513.699,E2 -3513.699} C_VEL
LIN {X 0,Y 544.618,Z 657.169,A -85,B 0,C 180,E1 -3515.183,E2 -3515.183} C_VEL
LIN {X 0,Y 544.692,Z 653.25,A -85,B 0,C 180,E1 -3516.668,E2 -3516.668} C_VEL
LIN {X 0,Y 544.736,Z 648.219,A -85,B 0,C 180,E1 -3518.159,E2 -3518.159} C_VEL
LIN {X 0,Y 544.792,Z 642.064,A -85,B 0,C 180,E1 -3519.654,E2 -3519.654} C_VEL
LIN {X 0,Y 545.003,Z 634.509,A -85,B 0,C 180,E1 -3521.153,E2 -3521.153} C_VEL
LIN {X 0,Y 545.192,Z 625.501,A -85,B 0,C 180,E1 -3522.659,E2 -3522.659} C_VEL
LIN {X 0,Y 545.517,Z 614.772,A -85,B 0,C 180,E1 -3524.169,E2 -3524.169} C_VEL
LIN {X 0,Y 545.87,Z 603.881,A -85,B 0,C 180,E1 -3525.476,E2 -3525.476} C_VEL
LIN {X 0,Y 546.312,Z 590.604,A -85,B 0,C 180,E1 -3526.825,E2 -3526.825} C_VEL
LIN {X 0,Y 546.819,Z 576.182,A -85,B 0,C 180,E1 -3528.053,E2 -3528.053} C_VEL
LIN {X 0,Y 547.277,Z 562.651,A -85,B 0,C 180,E1 -3529.017,E2 -3529.017} C_VEL
LIN {X 0,Y 547.722,Z 548.325,A -85,B 0,C 180,E1 -3529.879,E2 -3529.879} C_VEL
LIN {X 0,Y 548.13,Z 533.657,A -85,B 0,C 180,E1 -3530.612,E2 -3530.612} C_VEL
LIN {X 0,Y 548.585,Z 518.33,A -85,B 0,C 180,E1 -3531.218,E2 -3531.218} C_VEL
LIN {X 0,Y 548.898,Z 502.329,A -85,B 0,C 180,E1 -3531.698,E2 -3531.698} C_VEL
LIN {X 0,Y 549.124,Z 486.341,A -85,B 0,C 180,E1 -3532.034,E2 -3532.034} C_VEL
LIN {X 0,Y 550.277,Z 294.529,A -85,B 0,C 180,E1 -3534.673,E2 -3534.673} C_VEL
LIN {X 0,Y 548.052,Z 283.248,A -85,B 0,C 180,E1 -3534.951,E2 -3534.951} C_VEL
LIN {X 0,Y 547.928,Z 277.424,A -85,B 0,C 180,E1 -3535.572,E2 -3535.572} C_VEL
LIN {X 0,Y 545.108,Z 266.9,A -85,B 0,C 180,E1 -3536.867,E2 -3536.867} C_VEL
LIN {X 0,Y 545.059,Z 266.902,A -85,B 0,C 180,E1 -3539.338,E2 -3539.338} C_VEL
LIN {X 0,Y 545.054,Z 266.901,A -85,B 0,C 180,E1 -3541.915,E2 -3541.915} C_VEL
LIN {X 0,Y 545.06,Z 266.901,A -85,B 0,C 180,E1 -3544.564,E2 -3544.564} C_VEL
LIN {X 0,Y 545.03,Z 266.904,A -85,B 0,C 180,E1 -3547.304,E2 -3547.304} C_VEL
LIN {X 0,Y 545.064,Z 266.897,A -85,B 0,C 180,E1 -3550.142,E2 -3550.142} C_VEL
LIN {X 0,Y 545.085,Z 266.9,A -85,B 0,C 180,E1 -3553.105,E2 -3553.105} C_VEL
LIN {X 0,Y 545.049,Z 266.898,A -85,B 0,C 180,E1 -3556.226,E2 -3556.226} C_VEL
LIN {X 0,Y 545.084,Z 266.898,A -85,B 0,C 180,E1 -3558.886,E2 -3558.886} C_VEL
LIN {X 0,Y 545.05,Z 266.899,A -85,B 0,C 180,E1 -3561.762,E2 -3561.762} C_VEL
LIN {X 0,Y 545.052,Z 266.899,A -85,B 0,C 180,E1 -3564.533,E2 -3564.533} C_VEL
LIN {X 0,Y 545.066,Z 266.901,A -85,B 0,C 180,E1 -3567.211,E2 -3567.211} C_VEL
LIN {X 0,Y 545.062,Z 266.899,A -85,B 0,C 180,E1 -3569.81,E2 -3569.81} C_VEL
LIN {X 0,Y 545.078,Z 266.891,A -85,B 0,C 180,E1 -3572.344,E2 -3572.344} C_VEL
LIN {X 0,Y 545.115,Z 266.895,A -85,B 0,C 180,E1 -3574.82,E2 -3574.82} C_VEL
LIN {X 0,Y 545.042,Z 266.901,A -85,B 0,C 180,E1 -3577.242,E2 -3577.242} C_VEL
LIN {X 0,Y 545.113,Z 266.891,A -85,B 0,C 180,E1 -3580.415,E2 -3580.415} C_VEL
LIN {X 0,Y 545.07,Z 266.893,A -85,B 0,C 180,E1 -3583.521,E2 -3583.521} C_VEL
LIN {X 0,Y 545.092,Z 266.893,A -85,B 0,C 180,E1 -3585.82,E2 -3585.82} C_VEL
LIN {X 0,Y 545.116,Z 266.896,A -85,B 0,C 180,E1 -3588.849,E2 -3588.849} C_VEL
LIN {X 0,Y 545.125,Z 266.888,A -85,B 0,C 180,E1 -3591.847,E2 -3591.847} C_VEL
LIN {X 0,Y 545.204,Z 266.886,A -85,B 0,C 180,E1 -3594.823,E2 -3594.823} C_VEL
LIN {X 0,Y 545.195,Z 266.876,A -85,B 0,C 180,E1 -3597.784,E2 -3597.784} C_VEL
LIN {X 0,Y 545.21,Z 266.884,A -85,B 0,C 180,E1 -3600.738,E2 -3600.738} C_VEL
LIN {X 0,Y 545.169,Z 266.887,A -85,B 0,C 180,E1 -3602.956,E2 -3602.956} C_VEL
LIN {X 0,Y 545.176,Z 266.882,A -85,B 0,C 180,E1 -3605.919,E2 -3605.919} C_VEL
LIN {X 0,Y 545.114,Z 266.897,A -85,B 0,C 180,E1 -3608.9,E2 -3608.9} C_VEL
LIN {X 0,Y 545.132,Z 266.886,A -85,B 0,C 180,E1 -3611.904,E2 -3611.904} C_VEL
LIN {X 0,Y 545.083,Z 266.902,A -85,B 0,C 180,E1 -3614.944,E2 -3614.944} C_VEL
LIN {X 0,Y 545.076,Z 266.895,A -85,B 0,C 180,E1 -3618.026,E2 -3618.026} C_VEL
LIN {X 0,Y 545.092,Z 266.896,A -85,B 0,C 180,E1 -3620.372,E2 -3620.372} C_VEL
LIN {X 0,Y 545.088,Z 266.895,A -85,B 0,C 180,E1 -3623.559,E2 -3623.559} C_VEL
LIN {X 0,Y 545.076,Z 266.897,A -85,B 0,C 180,E1 -3626.001,E2 -3626.001} C_VEL
LIN {X 0,Y 545.086,Z 266.903,A -85,B 0,C 180,E1 -3628.748,E2 -3628.748} C_VEL
LIN {X 0,Y 545.055,Z 266.9,A -85,B 0,C 180,E1 -3631.679,E2 -3631.679} C_VEL
LIN {X 0,Y 545.079,Z 266.902,A -85,B 0,C 180,E1 -3634.563,E2 -3634.563} C_VEL
LIN {X 0,Y 545.036,Z 266.904,A -85,B 0,C 180,E1 -3637.304,E2 -3637.304} C_VEL
LIN {X 0,Y 545.069,Z 266.899,A -85,B 0,C 180,E1 -3640.142,E2 -3640.142} C_VEL
LIN {X 0,Y 545.06,Z 266.907,A -85,B 0,C 180,E1 -3642.697,E2 -3642.697} C_VEL
LIN {X 0,Y 545.056,Z 266.899,A -85,B 0,C 180,E1 -3645.871,E2 -3645.871} C_VEL
LIN {X 0,Y 545.095,Z 266.901,A -85,B 0,C 180,E1 -3648.887,E2 -3648.887} C_VEL
LIN {X 0,Y 545.05,Z 266.9,A -85,B 0,C 180,E1 -3651.763,E2 -3651.763} C_VEL
LIN {X 0,Y 545.034,Z 266.909,A -85,B 0,C 180,E1 -3654.532,E2 -3654.532} C_VEL
LIN {X 0,Y 545.066,Z 266.901,A -85,B 0,C 180,E1 -3657.212,E2 -3657.212} C_VEL
LIN {X 0,Y 545.062,Z 266.901,A -85,B 0,C 180,E1 -3659.811,E2 -3659.811} C_VEL
LIN {X 0,Y 545.072,Z 266.937,A -85,B 0,C 180,E1 -3660.798,E2 -3660.798} C_VEL
LIN {X 0,Y 548.833,Z 279.597,A -85,B 0,C 180,E1 -3662.19,E2 -3662.19} C_VEL
LIN {X 0,Y 548.808,Z 287.928,A -85,B 0,C 180,E1 -3662.96,E2 -3662.96} C_VEL
LIN {X 0,Y 548.246,Z 311.999,A -85,B 0,C 180,E1 -3665.109,E2 -3665.109} C_VEL
LIN {X 0,Y 550.262,Z 323.347,A -85,B 0,C 180,E1 -3665.365,E2 -3665.365} C_VEL
LIN {X 0,Y 549.085,Z 517.851,A -85,B 0,C 180,E1 -3668.039,E2 -3668.039} C_VEL
LIN {X 0,Y 548.839,Z 534.116,A -85,B 0,C 180,E1 -3668.399,E2 -3668.399} C_VEL
LIN {X 0,Y 548.48,Z 550.921,A -85,B 0,C 180,E1 -3668.926,E2 -3668.926} C_VEL
LIN {X 0,Y 548.104,Z 566.234,A -85,B 0,C 180,E1 -3669.555,E2 -3669.555} C_VEL
LIN {X 0,Y 547.654,Z 581.044,A -85,B 0,C 180,E1 -3670.314,E2 -3670.314} C_VEL
LIN {X 0,Y 547.153,Z 596.271,A -85,B 0,C 180,E1 -3671.27,E2 -3671.27} C_VEL
LIN {X 0,Y 546.63,Z 610.209,A -85,B 0,C 180,E1 -3672.317,E2 -3672.317} C_VEL
LIN {X 0,Y 546.157,Z 624.066,A -85,B 0,C 180,E1 -3673.555,E2 -3673.555} C_VEL
LIN {X 0,Y 545.837,Z 635.333,A -85,B 0,C 180,E1 -3674.734,E2 -3674.734} C_VEL
LIN {X 0,Y 545.467,Z 645.906,A -85,B 0,C 180,E1 -3676.02,E2 -3676.02} C_VEL
LIN {X 0,Y 545.182,Z 656.44,A -85,B 0,C 180,E1 -3677.53,E2 -3677.53} C_VEL
LIN {X 0,Y 544.957,Z 665.276,A -85,B 0,C 180,E1 -3679.034,E2 -3679.034} C_VEL
LIN {X 0,Y 544.795,Z 671.856,A -85,B 0,C 180,E1 -3680.346,E2 -3680.346} C_VEL
LIN {X 0,Y 544.739,Z 679.466,A -85,B 0,C 180,E1 -3682.214,E2 -3682.214} C_VEL
LIN {X 0,Y 544.686,Z 685.249,A -85,B 0,C 180,E1 -3684.075,E2 -3684.075} C_VEL
LIN {X 0,Y 544.6,Z 688.635,A -85,B 0,C 180,E1 -3685.559,E2 -3685.559} C_VEL
LIN {X 0,Y 544.638,Z 691.09,A -85,B 0,C 180,E1 -3687.041,E2 -3687.041} C_VEL
LIN {X 0,Y 544.539,Z 692.479,A -85,B 0,C 180,E1 -3688.521,E2 -3688.521} C_VEL
LIN {X 0,Y 544.536,Z 693,A -85,B 0,C 180,E1 -3690,E2 -3690} C_VEL
LIN {X 0,Y 544.539,Z 692.479,A -85,B 0,C 180,E1 -3691.479,E2 -3691.479} C_VEL
LIN {X 0,Y 544.638,Z 691.089,A -85,B 0,C 180,E1 -3692.959,E2 -3692.959} C_VEL
LIN {X 0,Y 544.6,Z 688.634,A -85,B 0,C 180,E1 -3694.441,E2 -3694.441} C_VEL
LIN {X 0,Y 544.686,Z 685.251,A -85,B 0,C 180,E1 -3695.925,E2 -3695.925} C_VEL
LIN {X 0,Y 544.739,Z 679.468,A -85,B 0,C 180,E1 -3697.786,E2 -3697.786} C_VEL
LIN {X 0,Y 544.795,Z 671.856,A -85,B 0,C 180,E1 -3699.654,E2 -3699.654} C_VEL
LIN {X 0,Y 545.017,Z 664.268,A -85,B 0,C 180,E1 -3701.153,E2 -3701.153} C_VEL
LIN {X 0,Y 545.228,Z 655.209,A -85,B 0,C 180,E1 -3702.658,E2 -3702.658} C_VEL
LIN {X 0,Y 545.529,Z 644.421,A -85,B 0,C 180,E1 -3704.168,E2 -3704.168} C_VEL
LIN {X 0,Y 545.926,Z 633.286,A -85,B 0,C 180,E1 -3705.493,E2 -3705.493} C_VEL
LIN {X 0,Y 546.263,Z 621.139,A -85,B 0,C 180,E1 -3706.73,E2 -3706.73} C_VEL
LIN {X 0,Y 546.72,Z 608.354,A -85,B 0,C 180,E1 -3707.833,E2 -3707.833} C_VEL
LIN {X 0,Y 547.153,Z 594.842,A -85,B 0,C 180,E1 -3708.828,E2 -3708.828} C_VEL
LIN {X 0,Y 547.649,Z 581.036,A -85,B 0,C 180,E1 -3709.686,E2 -3709.686} C_VEL
LIN {X 0,Y 548.126,Z 565.135,A -85,B 0,C 180,E1 -3710.498,E2 -3710.498} C_VEL
LIN {X 0,Y 548.53,Z 549.618,A -85,B 0,C 180,E1 -3711.121,E2 -3711.121} C_VEL
LIN {X 0,Y 548.874,Z 534.121,A -85,B 0,C 180,E1 -3711.6,E2 -3711.6} C_VEL
LIN {X 0,Y 549.091,Z 517.849,A -85,B 0,C 180,E1 -3711.961,E2 -3711.961} C_VEL
LIN {X 0,Y 550.215,Z 322.386,A -85,B 0,C 180,E1 -3714.65,E2 -3714.65} C_VEL
LIN {X 0,Y 548.194,Z 311.567,A -85,B 0,C 180,E1 -3714.905,E2 -3714.905} C_VEL
LIN {X 0,Y 549.001,Z 281.32,A -85,B 0,C 180,E1 -3717.641,E2 -3717.641} C_VEL
LIN {X 0,Y 548.34,Z 277.915,A -85,B 0,C 180,E1 -3717.992,E2 -3717.992} C_VEL
LIN {X 0,Y 545.082,Z 266.904,A -85,B 0,C 180,E1 -3719.221,E2 -3719.221} C_VEL
LIN {X 0,Y 545.053,Z 266.903,A -85,B 0,C 180,E1 -3721.915,E2 -3721.915} C_VEL
LIN {X 0,Y 545.06,Z 266.9,A -85,B 0,C 180,E1 -3724.564,E2 -3724.564} C_VEL
LIN {X 0,Y 545.035,Z 266.91,A -85,B 0,C 180,E1 -3727.304,E2 -3727.304} C_VEL
LIN {X 0,Y 545.067,Z 266.898,A -85,B 0,C 180,E1 -3730.142,E2 -3730.142} C_VEL
LIN {X 0,Y 545.084,Z 266.901,A -85,B 0,C 180,E1 -3733.106,E2 -3733.106} C_VEL
LIN {X 0,Y 545.047,Z 266.898,A -85,B 0,C 180,E1 -3736.226,E2 -3736.226} C_VEL
LIN {X 0,Y 545.095,Z 266.896,A -85,B 0,C 180,E1 -3738.887,E2 -3738.887} C_VEL
LIN {X 0,Y 545.049,Z 266.899,A -85,B 0,C 180,E1 -3741.763,E2 -3741.763} C_VEL
LIN {X 0,Y 545.051,Z 266.898,A -85,B 0,C 180,E1 -3744.533,E2 -3744.533} C_VEL
LIN {X 0,Y 545.066,Z 266.904,A -85,B 0,C 180,E1 -3747.212,E2 -3747.212} C_VEL
LIN {X 0,Y 545.061,Z 266.898,A -85,B 0,C 180,E1 -3749.81,E2 -3749.81} C_VEL
LIN {X 0,Y 545.078,Z 266.895,A -85,B 0,C 180,E1 -3752.344,E2 -3752.344} C_VEL
LIN {X 0,Y 545.115,Z 266.895,A -85,B 0,C 180,E1 -3754.82,E2 -3754.82} C_VEL
LIN {X 0,Y 545.042,Z 266.907,A -85,B 0,C 180,E1 -3757.243,E2 -3757.243} C_VEL
LIN {X 0,Y 545.113,Z 266.885,A -85,B 0,C 180,E1 -3760.415,E2 -3760.415} C_VEL
LIN {X 0,Y 545.07,Z 266.899,A -85,B 0,C 180,E1 -3763.521,E2 -3763.521} C_VEL
LIN {X 0,Y 545.092,Z 266.888,A -85,B 0,C 180,E1 -3765.82,E2 -3765.82} C_VEL
LIN {X 0,Y 545.116,Z 266.894,A -85,B 0,C 180,E1 -3768.849,E2 -3768.849} C_VEL
LIN {X 0,Y 545.126,Z 266.887,A -85,B 0,C 180,E1 -3771.847,E2 -3771.847} C_VEL
LIN {X 0,Y 545.204,Z 266.879,A -85,B 0,C 180,E1 -3774.823,E2 -3774.823} C_VEL
LIN {X 0,Y 545.196,Z 266.881,A -85,B 0,C 180,E1 -3777.784,E2 -3777.784} C_VEL
LIN {X 0,Y 545.209,Z 266.878,A -85,B 0,C 180,E1 -3780.739,E2 -3780.739} C_VEL
LIN {X 0,Y 545.169,Z 266.888,A -85,B 0,C 180,E1 -3782.956,E2 -3782.956} C_VEL
LIN {X 0,Y 545.169,Z 266.882,A -85,B 0,C 180,E1 -3785.92,E2 -3785.92} C_VEL
LIN {X 0,Y 545.115,Z 266.89,A -85,B 0,C 180,E1 -3788.9,E2 -3788.9} C_VEL
LIN {X 0,Y 545.133,Z 266.888,A -85,B 0,C 180,E1 -3791.904,E2 -3791.904} C_VEL
LIN {X 0,Y 545.084,Z 266.896,A -85,B 0,C 180,E1 -3794.944,E2 -3794.944} C_VEL
LIN {X 0,Y 545.076,Z 266.895,A -85,B 0,C 180,E1 -3798.026,E2 -3798.026} C_VEL
LIN {X 0,Y 545.093,Z 266.894,A -85,B 0,C 180,E1 -3800.372,E2 -3800.372} C_VEL
LIN {X 0,Y 545.09,Z 266.894,A -85,B 0,C 180,E1 -3803.559,E2 -3803.559} C_VEL
LIN {X 0,Y 545.077,Z 266.895,A -85,B 0,C 180,E1 -3806.001,E2 -3806.001} C_VEL
LIN {X 0,Y 545.087,Z 266.895,A -85,B 0,C 180,E1 -3808.748,E2 -3808.748} C_VEL
LIN {X 0,Y 545.056,Z 266.897,A -85,B 0,C 180,E1 -3811.679,E2 -3811.679} C_VEL
LIN {X 0,Y 545.08,Z 266.899,A -85,B 0,C 180,E1 -3814.563,E2 -3814.563} C_VEL
LIN {X 0,Y 545.065,Z 266.9,A -85,B 0,C 180,E1 -3817.002,E2 -3817.002} C_VEL
LIN {X 0,Y 544.355,Z 266.983,A -85,B 0,C 180,E1 -3817.618,E2 -3817.618} C_VEL
LIN {X 0,Y 541.488,Z 267.343,A -85,B 0,C 180,E1 -3818.619,E2 -3818.619} C_VEL
LIN {X 0,Y 539.1,Z 267.641,A -85,B 0,C 180,E1 -3819.425,E2 -3819.425} C_VEL
LIN {X 0,Y 538.091,Z 267.766,A -85,B 0,C 180,E1 -3820.047,E2 -3820.047} C_VEL
LIN {X 0,Y 538.015,Z 267.776,A -85,B 0,C 180,E1 -3820.257,E2 -3820.257} C_VEL
LIN {X 0,Y 538.025,Z 267.78,A -85,B 0,C 180,E1 -3822.988,E2 -3822.988} C_VEL
LIN {X 0,Y 538.025,Z 267.771,A -85,B 0,C 180,E1 -3825.926,E2 -3825.926} C_VEL
LIN {X 0,Y 538.051,Z 267.774,A -85,B 0,C 180,E1 -3829.225,E2 -3829.225} C_VEL
LIN {X 0,Y 537.992,Z 267.777,A -85,B 0,C 180,E1 -3832.123,E2 -3832.123} C_VEL
LIN {X 0,Y 537.997,Z 267.785,A -85,B 0,C 180,E1 -3834.916,E2 -3834.916} C_VEL
LIN {X 0,Y 538.018,Z 267.776,A -85,B 0,C 180,E1 -3837.618,E2 -3837.618} C_VEL
LIN {X 0,Y 538.015,Z 267.781,A -85,B 0,C 180,E1 -3840.239,E2 -3840.239} C_VEL
LIN {X 0,Y 538.069,Z 267.918,A -85,B 0,C 180,E1 -3842.954,E2 -3842.954} C_VEL
LIN {X 0,Y 541.399,Z 280.328,A -85,B 0,C 180,E1 -3844.477,E2 -3844.477} C_VEL
LIN {X 0,Y 541.4,Z 283.528,A -85,B 0,C 180,E1 -3844.819,E2 -3844.819} C_VEL
LIN {X 0,Y 543.864,Z 295.865,A -85,B 0,C 180,E1 -3845.123,E2 -3845.123} C_VEL
LIN {X 0,Y 542.515,Z 488.626,A -85,B 0,C 180,E1 -3847.809,E2 -3847.809} C_VEL
LIN {X 0,Y 542.253,Z 504.711,A -85,B 0,C 180,E1 -3848.173,E2 -3848.173} C_VEL
LIN {X 0,Y 541.865,Z 521.368,A -85,B 0,C 180,E1 -3848.706,E2 -3848.706} C_VEL
LIN {X 0,Y 541.404,Z 537.43,A -85,B 0,C 180,E1 -3849.384,E2 -3849.384} C_VEL
LIN {X 0,Y 540.917,Z 552.16,A -85,B 0,C 180,E1 -3850.158,E2 -3850.158} C_VEL
LIN {X 0,Y 540.335,Z 567.155,A -85,B 0,C 180,E1 -3851.123,E2 -3851.123} C_VEL
LIN {X 0,Y 539.827,Z 580.103,A -85,B 0,C 180,E1 -3852.12,E2 -3852.12} C_VEL
LIN {X 0,Y 539.27,Z 593.612,A -85,B 0,C 180,E1 -3853.339,E2 -3853.339} C_VEL
LIN {X 0,Y 538.904,Z 604.629,A -85,B 0,C 180,E1 -3854.494,E2 -3854.494} C_VEL
LIN {X 0,Y 538.515,Z 615.559,A -85,B 0,C 180,E1 -3855.836,E2 -3855.836} C_VEL
LIN {X 0,Y 538.217,Z 624.919,A -85,B 0,C 180,E1 -3857.174,E2 -3857.174} C_VEL
LIN {X 0,Y 537.98,Z 634.03,A -85,B 0,C 180,E1 -3858.7,E2 -3858.7} C_VEL
LIN {X 0,Y 537.745,Z 641.642,A -85,B 0,C 180,E1 -3860.218,E2 -3860.218} C_VEL
LIN {X 0,Y 537.669,Z 647.88,A -85,B 0,C 180,E1 -3861.733,E2 -3861.733} C_VEL
LIN {X 0,Y 537.6,Z 653.678,A -85,B 0,C 180,E1 -3863.484,E2 -3863.484} C_VEL
LIN {X 0,Y 537.545,Z 656.955,A -85,B 0,C 180,E1 -3864.749,E2 -3864.749} C_VEL
LIN {X 0,Y 537.56,Z 659.91,A -85,B 0,C 180,E1 -3866.252,E2 -3866.252} C_VEL
LIN {X 0,Y 537.485,Z 661.848,A -85,B 0,C 180,E1 -3867.752,E2 -3867.752} C_VEL
LIN {X 0,Y 537.437,Z 662.838,A -85,B 0,C 180,E1 -3869.251,E2 -3869.251} C_VEL
LIN {X 0,Y 537.437,Z 662.858,A -85,B 0,C 180,E1 -3870.749,E2 -3870.749} C_VEL
LIN {X 0,Y 537.485,Z 661.944,A -85,B 0,C 180,E1 -3872.248,E2 -3872.248} C_VEL
LIN {X 0,Y 537.559,Z 660.046,A -85,B 0,C 180,E1 -3873.748,E2 -3873.748} C_VEL
LIN {X 0,Y 537.543,Z 657.168,A -85,B 0,C 180,E1 -3875.251,E2 -3875.251} C_VEL
LIN {X 0,Y 537.616,Z 653.248,A -85,B 0,C 180,E1 -3876.757,E2 -3876.757} C_VEL
LIN {X 0,Y 537.661,Z 648.216,A -85,B 0,C 180,E1 -3878.267,E2 -3878.267} C_VEL
LIN {X 0,Y 537.737,Z 642.061,A -85,B 0,C 180,E1 -3879.782,E2 -3879.782} C_VEL
LIN {X 0,Y 538.021,Z 633.103,A -85,B 0,C 180,E1 -3881.564,E2 -3881.564} C_VEL
LIN {X 0,Y 538.21,Z 624.264,A -85,B 0,C 180,E1 -3883.018,E2 -3883.018} C_VEL
LIN {X 0,Y 538.56,Z 614.767,A -85,B 0,C 180,E1 -3884.356,E2 -3884.356} C_VEL
LIN {X 0,Y 538.927,Z 603.698,A -85,B 0,C 180,E1 -3885.7,E2 -3885.7} C_VEL
LIN {X 0,Y 539.433,Z 590.599,A -85,B 0,C 180,E1 -3887.046,E2 -3887.046} C_VEL
LIN {X 0,Y 540.013,Z 576.116,A -85,B 0,C 180,E1 -3888.299,E2 -3888.299} C_VEL
LIN {X 0,Y 540.529,Z 562.777,A -85,B 0,C 180,E1 -3889.264,E2 -3889.264} C_VEL
LIN {X 0,Y 541.031,Z 548.516,A -85,B 0,C 180,E1 -3890.135,E2 -3890.135} C_VEL
LIN {X 0,Y 541.492,Z 533.675,A -85,B 0,C 180,E1 -3890.884,E2 -3890.884} C_VEL
LIN {X 0,Y 541.987,Z 518.521,A -85,B 0,C 180,E1 -3891.489,E2 -3891.489} C_VEL
LIN {X 0,Y 542.303,Z 502.513,A -85,B 0,C 180,E1 -3891.975,E2 -3891.975} C_VEL
LIN {X 0,Y 542.561,Z 486.51,A -85,B 0,C 180,E1 -3892.315,E2 -3892.315} C_VEL
LIN {X 0,Y 543.838,Z 295.511,A -85,B 0,C 180,E1 -3894.974,E2 -3894.974} C_VEL
LIN {X 0,Y 541.392,Z 283.496,A -85,B 0,C 180,E1 -3895.275,E2 -3895.275} C_VEL
LIN {X 0,Y 541.256,Z 279.516,A -85,B 0,C 180,E1 -3895.706,E2 -3895.706} C_VEL
LIN {X 0,Y 538.051,Z 267.78,A -85,B 0,C 180,E1 -3897.178,E2 -3897.178} C_VEL
LIN {X 0,Y 538.013,Z 267.778,A -85,B 0,C 180,E1 -3899.761,E2 -3899.761} C_VEL
LIN {X 0,Y 538.018,Z 267.776,A -85,B 0,C 180,E1 -3902.382,E2 -3902.382} C_VEL
LIN {X 0,Y 537.994,Z 267.787,A -85,B 0,C 180,E1 -3905.084,E2 -3905.084} C_VEL
LIN {X 0,Y 537.988,Z 267.781,A -85,B 0,C 180,E1 -3907.878,E2 -3907.878} C_VEL
LIN {X 0,Y 538.047,Z 267.773,A -85,B 0,C 180,E1 -3910.775,E2 -3910.775} C_VEL
LIN {X 0,Y 538.028,Z 267.774,A -85,B 0,C 180,E1 -3914.074,E2 -3914.074} C_VEL
LIN {X 0,Y 538.018,Z 267.783,A -85,B 0,C 180,E1 -3917.214,E2 -3917.214} C_VEL
LIN {X 0,Y 538.021,Z 267.774,A -85,B 0,C 180,E1 -3920.203,E2 -3920.203} C_VEL
LIN {X 0,Y 538.025,Z 267.778,A -85,B 0,C 180,E1 -3923.067,E2 -3923.067} C_VEL
LIN {X 0,Y 538.022,Z 267.775,A -85,B 0,C 180,E1 -3925.827,E2 -3925.827} C_VEL
LIN {X 0,Y 538.006,Z 267.775,A -85,B 0,C 180,E1 -3928.498,E2 -3928.498} C_VEL
LIN {X 0,Y 538.058,Z 267.776,A -85,B 0,C 180,E1 -3931.1,E2 -3931.1} C_VEL
LIN {X 0,Y 538.039,Z 267.774,A -85,B 0,C 180,E1 -3933.633,E2 -3933.633} C_VEL
LIN {X 0,Y 538.021,Z 267.774,A -85,B 0,C 180,E1 -3936.118,E2 -3936.118} C_VEL
LIN {X 0,Y 538.035,Z 267.778,A -85,B 0,C 180,E1 -3939.348,E2 -3939.348} C_VEL
LIN {X 0,Y 538.052,Z 267.771,A -85,B 0,C 180,E1 -3942.517,E2 -3942.517} C_VEL
LIN {X 0,Y 538.061,Z 267.77,A -85,B 0,C 180,E1 -3945.631,E2 -3945.631} C_VEL
LIN {X 0,Y 538.075,Z 267.771,A -85,B 0,C 180,E1 -3948.701,E2 -3948.701} C_VEL
LIN {X 0,Y 538.082,Z 267.765,A -85,B 0,C 180,E1 -3951.739,E2 -3951.739} C_VEL
LIN {X 0,Y 538.162,Z 267.762,A -85,B 0,C 180,E1 -3954.755,E2 -3954.755} C_VEL
LIN {X 0,Y 538.167,Z 267.752,A -85,B 0,C 180,E1 -3957.755,E2 -3957.755} C_VEL
LIN {X 0,Y 538.18,Z 267.76,A -85,B 0,C 180,E1 -3960.748,E2 -3960.748} C_VEL
LIN {X 0,Y 538.135,Z 267.762,A -85,B 0,C 180,E1 -3962.994,E2 -3962.994} C_VEL
LIN {X 0,Y 538.13,Z 267.759,A -85,B 0,C 180,E1 -3965.997,E2 -3965.997} C_VEL
LIN {X 0,Y 538.065,Z 267.772,A -85,B 0,C 180,E1 -3969.018,E2 -3969.018} C_VEL
LIN {X 0,Y 538.08,Z 267.765,A -85,B 0,C 180,E1 -3972.062,E2 -3972.062} C_VEL
LIN {X 0,Y 538.042,Z 267.777,A -85,B 0,C 180,E1 -3975.144,E2 -3975.144} C_VEL
LIN {X 0,Y 538.029,Z 267.774,A -85,B 0,C 180,E1 -3978.27,E2 -3978.27} C_VEL
LIN {X 0,Y 538.036,Z 267.779,A -85,B 0,C 180,E1 -3980.651,E2 -3980.651} C_VEL
LIN {X 0,Y 538.021,Z 267.774,A -85,B 0,C 180,E1 -3983.887,E2 -3983.887} C_VEL
LIN {X 0,Y 538.038,Z 267.776,A -85,B 0,C 180,E1 -3986.367,E2 -3986.367} C_VEL
LIN {X 0,Y 538.028,Z 267.782,A -85,B 0,C 180,E1 -3988.934,E2 -3988.934} C_VEL
LIN {X 0,Y 538.01,Z 267.777,A -85,B 0,C 180,E1 -3991.888,E2 -3991.888} C_VEL
LIN {X 0,Y 538.029,Z 267.782,A -85,B 0,C 180,E1 -3994.621,E2 -3994.621} C_VEL
LIN {X 0,Y 538.005,Z 267.782,A -85,B 0,C 180,E1 -3997.171,E2 -3997.171} C_VEL
LIN {X 0,Y 538.024,Z 267.776,A -85,B 0,C 180,E1 -3999.797,E2 -3999.797} C_VEL
LIN {X 0,Y 538.017,Z 267.785,A -85,B 0,C 180,E1 -4002.786,E2 -4002.786} C_VEL
LIN {X 0,Y 538.026,Z 267.775,A -85,B 0,C 180,E1 -4005.926,E2 -4005.926} C_VEL
LIN {X 0,Y 538.049,Z 267.775,A -85,B 0,C 180,E1 -4009.225,E2 -4009.225} C_VEL
LIN {X 0,Y 537.989,Z 267.781,A -85,B 0,C 180,E1 -4012.122,E2 -4012.122} C_VEL
LIN {X 0,Y 537.996,Z 267.778,A -85,B 0,C 180,E1 -4014.916,E2 -4014.916} C_VEL
LIN {X 0,Y 538.016,Z 267.777,A -85,B 0,C 180,E1 -4017.617,E2 -4017.617} C_VEL
LIN {X 0,Y 538.052,Z 267.924,A -85,B 0,C 180,E1 -4020.495,E2 -4020.495} C_VEL
LIN {X 0,Y 542.214,Z 281.843,A -85,B 0,C 180,E1 -4022.052,E2 -4022.052} C_VEL
LIN {X 0,Y 541.847,Z 299.117,A -85,B 0,C 180,E1 -4023.649,E2 -4023.649} C_VEL
LIN {X 0,Y 541.502,Z 311.325,A -85,B 0,C 180,E1 -4024.763,E2 -4024.763} C_VEL
LIN {X 0,Y 543.768,Z 323.478,A -85,B 0,C 180,E1 -4025.056,E2 -4025.056} C_VEL
LIN {X 0,Y 542.492,Z 517.643,A -85,B 0,C 180,E1 -4027.758,E2 -4027.758} C_VEL
LIN {X 0,Y 542.249,Z 533.909,A -85,B 0,C 180,E1 -4028.123,E2 -4028.123} C_VEL
LIN {X 0,Y 541.833,Z 550.713,A -85,B 0,C 180,E1 -4028.655,E2 -4028.655} C_VEL
LIN {X 0,Y 541.411,Z 566.057,A -85,B 0,C 180,E1 -4029.291,E2 -4029.291} C_VEL
LIN {X 0,Y 540.899,Z 580.925,A -85,B 0,C 180,E1 -4030.058,E2 -4030.058} C_VEL
LIN {X 0,Y 540.322,Z 596.225,A -85,B 0,C 180,E1 -4031.024,E2 -4031.024} C_VEL
LIN {X 0,Y 539.828,Z 609.242,A -85,B 0,C 180,E1 -4032.006,E2 -4032.006} C_VEL
LIN {X 0,Y 539.35,Z 622.114,A -85,B 0,C 180,E1 -4033.147,E2 -4033.147} C_VEL
LIN {X 0,Y 538.949,Z 633.285,A -85,B 0,C 180,E1 -4034.301,E2 -4034.301} C_VEL
LIN {X 0,Y 538.586,Z 644.421,A -85,B 0,C 180,E1 -4035.645,E2 -4035.645} C_VEL
LIN {X 0,Y 538.204,Z 655.207,A -85,B 0,C 180,E1 -4037.174,E2 -4037.174} C_VEL
LIN {X 0,Y 537.99,Z 664.268,A -85,B 0,C 180,E1 -4038.7,E2 -4038.7} C_VEL
LIN {X 0,Y 537.739,Z 671.856,A -85,B 0,C 180,E1 -4040.218,E2 -4040.218} C_VEL
LIN {X 0,Y 537.658,Z 679.465,A -85,B 0,C 180,E1 -4042.111,E2 -4042.111} C_VEL
LIN {X 0,Y 537.587,Z 685.249,A -85,B 0,C 180,E1 -4043.997,E2 -4043.997} C_VEL
LIN {X 0,Y 537.5,Z 688.635,A -85,B 0,C 180,E1 -4045.5,E2 -4045.5} C_VEL
LIN {X 0,Y 537.538,Z 691.091,A -85,B 0,C 180,E1 -4047.002,E2 -4047.002} C_VEL
LIN {X 0,Y 537.445,Z 692.479,A -85,B 0,C 180,E1 -4048.501,E2 -4048.501} C_VEL
LIN {X 0,Y 537.437,Z 693,A -85,B 0,C 180,E1 -4050,E2 -4050} C_VEL
LIN {X 0,Y 537.445,Z 692.478,A -85,B 0,C 180,E1 -4051.499,E2 -4051.499} C_VEL
LIN {X 0,Y 537.538,Z 691.089,A -85,B 0,C 180,E1 -4052.998,E2 -4052.998} C_VEL
LIN {X 0,Y 537.5,Z 688.634,A -85,B 0,C 180,E1 -4054.5,E2 -4054.5} C_VEL
LIN {X 0,Y 537.586,Z 685.252,A -85,B 0,C 180,E1 -4056.003,E2 -4056.003} C_VEL
LIN {X 0,Y 537.658,Z 679.468,A -85,B 0,C 180,E1 -4057.889,E2 -4057.889} C_VEL
LIN {X 0,Y 537.739,Z 671.856,A -85,B 0,C 180,E1 -4059.782,E2 -4059.782} C_VEL
LIN {X 0,Y 537.99,Z 664.268,A -85,B 0,C 180,E1 -4061.3,E2 -4061.3} C_VEL
LIN {X 0,Y 538.204,Z 655.208,A -85,B 0,C 180,E1 -4062.826,E2 -4062.826} C_VEL
LIN {X 0,Y 538.585,Z 644.421,A -85,B 0,C 180,E1 -4064.355,E2 -4064.355} C_VEL
LIN {X 0,Y 538.979,Z 633.285,A -85,B 0,C 180,E1 -4065.698,E2 -4065.698} C_VEL
LIN {X 0,Y 539.414,Z 621.137,A -85,B 0,C 180,E1 -4066.949,E2 -4066.949} C_VEL
LIN {X 0,Y 539.949,Z 607.733,A -85,B 0,C 180,E1 -4068.116,E2 -4068.116} C_VEL
LIN {X 0,Y 540.447,Z 593.356,A -85,B 0,C 180,E1 -4069.169,E2 -4069.169} C_VEL
LIN {X 0,Y 540.901,Z 579.143,A -85,B 0,C 180,E1 -4070.041,E2 -4070.041} C_VEL
LIN {X 0,Y 541.458,Z 563.747,A -85,B 0,C 180,E1 -4070.817,E2 -4070.817} C_VEL
LIN {X 0,Y 541.913,Z 548.107,A -85,B 0,C 180,E1 -4071.442,E2 -4071.442} C_VEL
LIN {X 0,Y 542.26,Z 532.076,A -85,B 0,C 180,E1 -4071.927,E2 -4071.927} C_VEL
LIN {X 0,Y 542.515,Z 516.134,A -85,B 0,C 180,E1 -4072.267,E2 -4072.267} C_VEL
LIN {X 0,Y 543.766,Z 323.517,A -85,B 0,C 180,E1 -4074.944,E2 -4074.944} C_VEL
LIN {X 0,Y 541.527,Z 311.118,A -85,B 0,C 180,E1 -4075.255,E2 -4075.255} C_VEL
LIN {X 0,Y 542.364,Z 283.27,A -85,B 0,C 180,E1 -4077.807,E2 -4077.807} C_VEL
LIN {X 0,Y 541.204,Z 278.58,A -85,B 0,C 180,E1 -4078.311,E2 -4078.311} C_VEL
LIN {X 0,Y 538.026,Z 267.782,A -85,B 0,C 180,E1 -4079.532,E2 -4079.532} C_VEL
LIN {X 0,Y 538.017,Z 267.778,A -85,B 0,C 180,E1 -4082.383,E2 -4082.383} C_VEL
LIN {X 0,Y 537.996,Z 267.785,A -85,B 0,C 180,E1 -4085.084,E2 -4085.084} C_VEL
LIN {X 0,Y 537.991,Z 267.781,A -85,B 0,C 180,E1 -4087.878,E2 -4087.878} C_VEL
LIN {X 0,Y 538.048,Z 267.775,A -85,B 0,C 180,E1 -4090.775,E2 -4090.775} C_VEL
LIN {X 0,Y 538.027,Z 267.773,A -85,B 0,C 180,E1 -4094.074,E2 -4094.074} C_VEL
LIN {X 0,Y 538.017,Z 267.782,A -85,B 0,C 180,E1 -4097.214,E2 -4097.214} C_VEL
LIN {X 0,Y 538.024,Z 267.772,A -85,B 0,C 180,E1 -4100.203,E2 -4100.203} C_VEL
LIN {X 0,Y 538.025,Z 267.779,A -85,B 0,C 180,E1 -4103.067,E2 -4103.067} C_VEL
LIN {X 0,Y 538.022,Z 267.775,A -85,B 0,C 180,E1 -4105.827,E2 -4105.827} C_VEL
LIN {X 0,Y 538.006,Z 267.777,A -85,B 0,C 180,E1 -4108.499,E2 -4108.499} C_VEL
LIN {X 0,Y 538.057,Z 267.777,A -85,B 0,C 180,E1 -4111.1,E2 -4111.1} C_VEL
LIN {X 0,Y 538.039,Z 267.775,A -85,B 0,C 180,E1 -4113.633,E2 -4113.633} C_VEL
LIN {X 0,Y 538.02,Z 267.774,A -85,B 0,C 180,E1 -4116.118,E2 -4116.118} C_VEL
LIN {X 0,Y 538.035,Z 267.771,A -85,B 0,C 180,E1 -4119.349,E2 -4119.349} C_VEL
LIN {X 0,Y 538.052,Z 267.771,A -85,B 0,C 180,E1 -4122.517,E2 -4122.517} C_VEL
LIN {X 0,Y 538.061,Z 267.765,A -85,B 0,C 180,E1 -4125.631,E2 -4125.631} C_VEL
LIN {X 0,Y 538.075,Z 267.769,A -85,B 0,C 180,E1 -4128.702,E2 -4128.702} C_VEL
LIN {X 0,Y 538.083,Z 267.764,A -85,B 0,C 180,E1 -4131.74,E2 -4131.74} C_VEL
LIN {X 0,Y 538.162,Z 267.754,A -85,B 0,C 180,E1 -4134.755,E2 -4134.755} C_VEL
LIN {X 0,Y 538.167,Z 267.756,A -85,B 0,C 180,E1 -4137.755,E2 -4137.755} C_VEL
LIN {X 0,Y 538.18,Z 267.753,A -85,B 0,C 180,E1 -4140.748,E2 -4140.748} C_VEL
LIN {X 0,Y 538.136,Z 267.765,A -85,B 0,C 180,E1 -4142.995,E2 -4142.995} C_VEL
LIN {X 0,Y 538.119,Z 267.76,A -85,B 0,C 180,E1 -4145.997,E2 -4145.997} C_VEL
LIN {X 0,Y 538.066,Z 267.769,A -85,B 0,C 180,E1 -4149.018,E2 -4149.018} C_VEL
LIN {X 0,Y 538.081,Z 267.767,A -85,B 0,C 180,E1 -4152.063,E2 -4152.063} C_VEL
LIN {X 0,Y 538.043,Z 267.771,A -85,B 0,C 180,E1 -4155.144,E2 -4155.144} C_VEL
LIN {X 0,Y 538.029,Z 267.774,A -85,B 0,C 180,E1 -4158.27,E2 -4158.27} C_VEL
LIN {X 0,Y 538.037,Z 267.776,A -85,B 0,C 180,E1 -4160.652,E2 -4160.652} C_VEL
LIN {X 0,Y 538.023,Z 267.773,A -85,B 0,C 180,E1 -4163.888,E2 -4163.888} C_VEL
LIN {X 0,Y 538.039,Z 267.773,A -85,B 0,C 180,E1 -4166.367,E2 -4166.367} C_VEL
LIN {X 0,Y 538.029,Z 267.777,A -85,B 0,C 180,E1 -4168.934,E2 -4168.934} C_VEL
LIN {X 0,Y 538.008,Z 267.775,A -85,B 0,C 180,E1 -4171.887,E2 -4171.887} C_VEL
LIN {X 0,Y 538.03,Z 267.778,A -85,B 0,C 180,E1 -4174.621,E2 -4174.621} C_VEL
LIN {X 0,Y 538.006,Z 267.776,A -85,B 0,C 180,E1 -4177.171,E2 -4177.171} C_VEL
LIN {X 0,Y 538.015,Z 267.776,A -85,B 0,C 180,E1 -4180.257,E2 -4180.257} C_VEL
LIN {X 0,Y 537.367,Z 267.862,A -85,B 0,C 180,E1 -4180.883,E2 -4180.883} C_VEL
LIN {X 0,Y 534.519,Z 268.218,A -85,B 0,C 180,E1 -4181.897,E2 -4181.897} C_VEL
LIN {X 0,Y 532.097,Z 268.517,A -85,B 0,C 180,E1 -4182.715,E2 -4182.715} C_VEL
LIN {X 0,Y 531.049,Z 268.646,A -85,B 0,C 180,E1 -4183.346,E2 -4183.346} C_VEL
LIN {X 0,Y 530.961,Z 268.655,A -85,B 0,C 180,E1 -4183.559,E2 -4183.559} C_VEL
LIN {X 0,Y 530.96,Z 268.655,A -85,B 0,C 180,E1 -4186.505,E2 -4186.505} C_VEL
LIN {X 0,Y 530.989,Z 268.658,A -85,B 0,C 180,E1 -4188.976,E2 -4188.976} C_VEL
LIN {X 0,Y 530.958,Z 268.653,A -85,B 0,C 180,E1 -4191.53,E2 -4191.53} C_VEL
LIN {X 0,Y 530.953,Z 268.657,A -85,B 0,C 180,E1 -4194.38,E2 -4194.38} C_VEL
LIN {X 0,Y 530.967,Z 268.653,A -85,B 0,C 180,E1 -4197.134,E2 -4197.134} C_VEL
LIN {X 0,Y 530.969,Z 268.656,A -85,B 0,C 180,E1 -4199.803,E2 -4199.803} C_VEL
LIN {X 0,Y 531.06,Z 268.845,A -85,B 0,C 180,E1 -4202.648,E2 -4202.648} C_VEL
LIN {X 0,Y 534.647,Z 282.026,A -85,B 0,C 180,E1 -4204.292,E2 -4204.292} C_VEL
LIN {X 0,Y 534.779,Z 283.801,A -85,B 0,C 180,E1 -4204.489,E2 -4204.489} C_VEL
LIN {X 0,Y 537.437,Z 297.502,A -85,B 0,C 180,E1 -4204.825,E2 -4204.825} C_VEL
LIN {X 0,Y 535.989,Z 487.367,A -85,B 0,C 180,E1 -4207.498,E2 -4207.498} C_VEL
LIN {X 0,Y 535.702,Z 504.027,A -85,B 0,C 180,E1 -4207.867,E2 -4207.867} C_VEL
LIN {X 0,Y 535.297,Z 520.297,A -85,B 0,C 180,E1 -4208.381,E2 -4208.381} C_VEL
LIN {X 0,Y 534.836,Z 535.67,A -85,B 0,C 180,E1 -4209.018,E2 -4209.018} C_VEL
LIN {X 0,Y 534.233,Z 550.646,A -85,B 0,C 180,E1 -4209.798,E2 -4209.798} C_VEL
LIN {X 0,Y 533.717,Z 564.534,A -85,B 0,C 180,E1 -4210.68,E2 -4210.68} C_VEL
LIN {X 0,Y 533.111,Z 578.737,A -85,B 0,C 180,E1 -4211.752,E2 -4211.752} C_VEL
LIN {X 0,Y 532.494,Z 591.85,A -85,B 0,C 180,E1 -4212.923,E2 -4212.923} C_VEL
LIN {X 0,Y 532.067,Z 602.978,A -85,B 0,C 180,E1 -4214.093,E2 -4214.093} C_VEL
LIN {X 0,Y 531.648,Z 614.097,A -85,B 0,C 180,E1 -4215.454,E2 -4215.454} C_VEL
LIN {X 0,Y 531.217,Z 624.921,A -85,B 0,C 180,E1 -4217.002,E2 -4217.002} C_VEL
LIN {X 0,Y 530.953,Z 634.032,A -85,B 0,C 180,E1 -4218.548,E2 -4218.548} C_VEL
LIN {X 0,Y 530.701,Z 641.645,A -85,B 0,C 180,E1 -4220.087,E2 -4220.087} C_VEL
LIN {X 0,Y 530.609,Z 647.882,A -85,B 0,C 180,E1 -4221.622,E2 -4221.622} C_VEL
LIN {X 0,Y 530.549,Z 652.998,A -85,B 0,C 180,E1 -4223.153,E2 -4223.153} C_VEL
LIN {X 0,Y 530.471,Z 656.956,A -85,B 0,C 180,E1 -4224.679,E2 -4224.679} C_VEL
LIN {X 0,Y 530.479,Z 659.91,A -85,B 0,C 180,E1 -4226.202,E2 -4226.202} C_VEL
LIN {X 0,Y 530.406,Z 661.848,A -85,B 0,C 180,E1 -4227.722,E2 -4227.722} C_VEL
LIN {X 0,Y 530.339,Z 662.838,A -85,B 0,C 180,E1 -4229.241,E2 -4229.241} C_VEL
LIN {X 0,Y 530.339,Z 662.857,A -85,B 0,C 180,E1 -4230.759,E2 -4230.759} C_VEL
LIN {X 0,Y 530.406,Z 661.944,A -85,B 0,C 180,E1 -4232.278,E2 -4232.278} C_VEL
LIN {X 0,Y 530.478,Z 660.044,A -85,B 0,C 180,E1 -4233.798,E2 -4233.798} C_VEL
LIN {X 0,Y 530.47,Z 657.166,A -85,B 0,C 180,E1 -4235.321,E2 -4235.321} C_VEL
LIN {X 0,Y 530.548,Z 653.246,A -85,B 0,C 180,E1 -4236.847,E2 -4236.847} C_VEL
LIN {X 0,Y 530.602,Z 648.214,A -85,B 0,C 180,E1 -4238.378,E2 -4238.378} C_VEL
LIN {X 0,Y 530.694,Z 642.059,A -85,B 0,C 180,E1 -4239.913,E2 -4239.913} C_VEL
LIN {X 0,Y 530.987,Z 633.531,A -85,B 0,C 180,E1 -4241.638,E2 -4241.638} C_VEL
LIN {X 0,Y 531.222,Z 624.259,A -85,B 0,C 180,E1 -4243.192,E2 -4243.192} C_VEL
LIN {X 0,Y 531.666,Z 613.591,A -85,B 0,C 180,E1 -4244.703,E2 -4244.703} C_VEL
LIN {X 0,Y 532.09,Z 602.021,A -85,B 0,C 180,E1 -4246.103,E2 -4246.103} C_VEL
LIN {X 0,Y 532.631,Z 589.724,A -85,B 0,C 180,E1 -4247.369,E2 -4247.369} C_VEL
LIN {X 0,Y 533.228,Z 576.317,A -85,B 0,C 180,E1 -4248.54,E2 -4248.54} C_VEL
LIN {X 0,Y 533.787,Z 562.976,A -85,B 0,C 180,E1 -4249.517,E2 -4249.517} C_VEL
LIN {X 0,Y 534.357,Z 548.712,A -85,B 0,C 180,E1 -4250.398,E2 -4250.398} C_VEL
LIN {X 0,Y 534.855,Z 533.931,A -85,B 0,C 180,E1 -4251.152,E2 -4251.152} C_VEL
LIN {X 0,Y 535.382,Z 518.712,A -85,B 0,C 180,E1 -4251.767,E2 -4251.767} C_VEL
LIN {X 0,Y 535.736,Z 502.697,A -85,B 0,C 180,E1 -4252.259,E2 -4252.259} C_VEL
LIN {X 0,Y 536.023,Z 486.678,A -85,B 0,C 180,E1 -4252.602,E2 -4252.602} C_VEL
LIN {X 0,Y 537.401,Z 296.619,A -85,B 0,C 180,E1 -4255.28,E2 -4255.28} C_VEL
LIN {X 0,Y 534.728,Z 283.616,A -85,B 0,C 180,E1 -4255.622,E2 -4255.622} C_VEL
LIN {X 0,Y 533.948,Z 279.285,A -85,B 0,C 180,E1 -4256.133,E2 -4256.133} C_VEL
LIN {X 0,Y 530.998,Z 268.657,A -85,B 0,C 180,E1 -4257.489,E2 -4257.489} C_VEL
LIN {X 0,Y 530.968,Z 268.656,A -85,B 0,C 180,E1 -4260.197,E2 -4260.197} C_VEL
LIN {X 0,Y 530.966,Z 268.654,A -85,B 0,C 180,E1 -4262.866,E2 -4262.866} C_VEL
LIN {X 0,Y 530.949,Z 268.655,A -85,B 0,C 180,E1 -4265.62,E2 -4265.62} C_VEL
LIN {X 0,Y 530.963,Z 268.656,A -85,B 0,C 180,E1 -4268.653,E2 -4268.653} C_VEL
LIN {X 0,Y 530.993,Z 268.656,A -85,B 0,C 180,E1 -4271.435,E2 -4271.435} C_VEL
LIN {X 0,Y 530.987,Z 268.652,A -85,B 0,C 180,E1 -4274.546,E2 -4274.546} C_VEL
LIN {X 0,Y 530.983,Z 268.652,A -85,B 0,C 180,E1 -4277.834,E2 -4277.834} C_VEL
LIN {X 0,Y 530.984,Z 268.652,A -85,B 0,C 180,E1 -4280.556,E2 -4280.556} C_VEL
LIN {X 0,Y 530.964,Z 268.659,A -85,B 0,C 180,E1 -4283.442,E2 -4283.442} C_VEL
LIN {X 0,Y 530.997,Z 268.649,A -85,B 0,C 180,E1 -4286.494,E2 -4286.494} C_VEL
LIN {X 0,Y 530.972,Z 268.659,A -85,B 0,C 180,E1 -4289.355,E2 -4289.355} C_VEL
LIN {X 0,Y 531.01,Z 268.643,A -85,B 0,C 180,E1 -4292.467,E2 -4292.467} C_VEL
LIN {X 0,Y 531.003,Z 268.654,A -85,B 0,C 180,E1 -4294.942,E2 -4294.942} C_VEL
LIN {X 0,Y 530.969,Z 268.646,A -85,B 0,C 180,E1 -4298.246,E2 -4298.246} C_VEL
LIN {X 0,Y 530.99,Z 268.653,A -85,B 0,C 180,E1 -4300.677,E2 -4300.677} C_VEL
LIN {X 0,Y 530.983,Z 268.653,A -85,B 0,C 180,E1 -4303.071,E2 -4303.071} C_VEL
LIN {X 0,Y 531.017,Z 268.65,A -85,B 0,C 180,E1 -4305.436,E2 -4305.436} C_VEL
LIN {X 0,Y 531.034,Z 268.647,A -85,B 0,C 180,E1 -4308.55,E2 -4308.55} C_VEL
LIN {X 0,Y 531.051,Z 268.642,A -85,B 0,C 180,E1 -4311.629,E2 -4311.629} C_VEL
LIN {X 0,Y 531.122,Z 268.638,A -85,B 0,C 180,E1 -4314.685,E2 -4314.685} C_VEL
LIN {X 0,Y 531.139,Z 268.627,A -85,B 0,C 180,E1 -4317.725,E2 -4317.725} C_VEL
LIN {X 0,Y 531.15,Z 268.636,A -85,B 0,C 180,E1 -4320.758,E2 -4320.758} C_VEL
LIN {X 0,Y 531.102,Z 268.636,A -85,B 0,C 180,E1 -4323.034,E2 -4323.034} C_VEL
LIN {X 0,Y 531.089,Z 268.637,A -85,B 0,C 180,E1 -4326.077,E2 -4326.077} C_VEL
LIN {X 0,Y 531.026,Z 268.647,A -85,B 0,C 180,E1 -4329.138,E2 -4329.138} C_VEL
LIN {X 0,Y 531.038,Z 268.642,A -85,B 0,C 180,E1 -4332.225,E2 -4332.225} C_VEL
LIN {X 0,Y 530.992,Z 268.653,A -85,B 0,C 180,E1 -4335.35,E2 -4335.35} C_VEL
LIN {X 0,Y 530.988,Z 268.654,A -85,B 0,C 180,E1 -4338.521,E2 -4338.521} C_VEL
LIN {X 0,Y 530.997,Z 268.657,A -85,B 0,C 180,E1 -4340.938,E2 -4340.938} C_VEL
LIN {X 0,Y 530.977,Z 268.653,A -85,B 0,C 180,E1 -4344.224,E2 -4344.224} C_VEL
LIN {X 0,Y 530.998,Z 268.659,A -85,B 0,C 180,E1 -4346.744,E2 -4346.744} C_VEL
LIN {X 0,Y 530.978,Z 268.655,A -85,B 0,C 180,E1 -4349.323,E2 -4349.323} C_VEL
LIN {X 0,Y 530.967,Z 268.656,A -85,B 0,C 180,E1 -4352.101,E2 -4352.101} C_VEL
LIN {X 0,Y 530.986,Z 268.66,A -85,B 0,C 180,E1 -4354.854,E2 -4354.854} C_VEL
LIN {X 0,Y 530.963,Z 268.656,A -85,B 0,C 180,E1 -4357.508,E2 -4357.508} C_VEL
LIN {X 0,Y 530.981,Z 268.658,A -85,B 0,C 180,E1 -4360.433,E2 -4360.433} C_VEL
LIN {X 0,Y 530.958,Z 268.658,A -85,B 0,C 180,E1 -4363.281,E2 -4363.281} C_VEL
LIN {X 0,Y 530.985,Z 268.652,A -85,B 0,C 180,E1 -4365.621,E2 -4365.621} C_VEL
LIN {X 0,Y 530.998,Z 268.657,A -85,B 0,C 180,E1 -4368.565,E2 -4368.565} C_VEL
LIN {X 0,Y 530.955,Z 268.656,A -85,B 0,C 180,E1 -4371.53,E2 -4371.53} C_VEL
LIN {X 0,Y 530.952,Z 268.662,A -85,B 0,C 180,E1 -4374.38,E2 -4374.38} C_VEL
LIN {X 0,Y 530.964,Z 268.658,A -85,B 0,C 180,E1 -4377.134,E2 -4377.134} C_VEL
LIN {X 0,Y 530.976,Z 268.716,A -85,B 0,C 180,E1 -4380.16,E2 -4380.16} C_VEL
LIN {X 0,Y 535.629,Z 284.421,A -85,B 0,C 180,E1 -4381.943,E2 -4381.943} C_VEL
LIN {X 0,Y 534.84,Z 311.257,A -85,B 0,C 180,E1 -4384.437,E2 -4384.437} C_VEL
LIN {X 0,Y 537.339,Z 325.459,A -85,B 0,C 180,E1 -4384.768,E2 -4384.768} C_VEL
LIN {X 0,Y 535.936,Z 517.436,A -85,B 0,C 180,E1 -4387.471,E2 -4387.471} C_VEL
LIN {X 0,Y 535.676,Z 532.783,A -85,B 0,C 180,E1 -4387.815,E2 -4387.815} C_VEL
LIN {X 0,Y 535.246,Z 547.895,A -85,B 0,C 180,E1 -4388.278,E2 -4388.278} C_VEL
LIN {X 0,Y 534.832,Z 563.332,A -85,B 0,C 180,E1 -4388.904,E2 -4388.904} C_VEL
LIN {X 0,Y 534.172,Z 578.942,A -85,B 0,C 180,E1 -4389.696,E2 -4389.696} C_VEL
LIN {X 0,Y 533.664,Z 593.149,A -85,B 0,C 180,E1 -4390.578,E2 -4390.578} C_VEL
LIN {X 0,Y 533.156,Z 606.496,A -85,B 0,C 180,E1 -4391.557,E2 -4391.557} C_VEL
LIN {X 0,Y 532.581,Z 620.001,A -85,B 0,C 180,E1 -4392.728,E2 -4392.728} C_VEL
LIN {X 0,Y 532.102,Z 631.469,A -85,B 0,C 180,E1 -4393.897,E2 -4393.897} C_VEL
LIN {X 0,Y 531.724,Z 642.032,A -85,B 0,C 180,E1 -4395.141,E2 -4395.141} C_VEL
LIN {X 0,Y 531.288,Z 652.74,A -85,B 0,C 180,E1 -4396.615,E2 -4396.615} C_VEL
LIN {X 0,Y 531.02,Z 662.094,A -85,B 0,C 180,E1 -4398.15,E2 -4398.15} C_VEL
LIN {X 0,Y 530.783,Z 670.048,A -85,B 0,C 180,E1 -4399.703,E2 -4399.703} C_VEL
LIN {X 0,Y 530.627,Z 676.624,A -85,B 0,C 180,E1 -4401.239,E2 -4401.239} C_VEL
LIN {X 0,Y 530.56,Z 681.957,A -85,B 0,C 180,E1 -4402.771,E2 -4402.771} C_VEL
LIN {X 0,Y 530.495,Z 685.25,A -85,B 0,C 180,E1 -4403.916,E2 -4403.916} C_VEL
LIN {X 0,Y 530.403,Z 688.634,A -85,B 0,C 180,E1 -4405.44,E2 -4405.44} C_VEL
LIN {X 0,Y 530.444,Z 691.091,A -85,B 0,C 180,E1 -4406.962,E2 -4406.962} C_VEL
LIN {X 0,Y 530.355,Z 692.478,A -85,B 0,C 180,E1 -4408.481,E2 -4408.481} C_VEL
LIN {X 0,Y 530.338,Z 693,A -85,B 0,C 180,E1 -4410,E2 -4410} C_VEL
LIN {X 0,Y 530.355,Z 692.478,A -85,B 0,C 180,E1 -4411.519,E2 -4411.519} C_VEL
LIN {X 0,Y 530.444,Z 691.089,A -85,B 0,C 180,E1 -4413.038,E2 -4413.038} C_VEL
LIN {X 0,Y 530.403,Z 688.633,A -85,B 0,C 180,E1 -4414.56,E2 -4414.56} C_VEL
LIN {X 0,Y 530.494,Z 685.252,A -85,B 0,C 180,E1 -4416.084,E2 -4416.084} C_VEL
LIN {X 0,Y 530.569,Z 679.468,A -85,B 0,C 180,E1 -4417.995,E2 -4417.995} C_VEL
LIN {X 0,Y 530.696,Z 671.856,A -85,B 0,C 180,E1 -4419.913,E2 -4419.913} C_VEL
LIN {X 0,Y 531,Z 663.252,A -85,B 0,C 180,E1 -4421.646,E2 -4421.646} C_VEL
LIN {X 0,Y 531.228,Z 653.976,A -85,B 0,C 180,E1 -4423.192,E2 -4423.192} C_VEL
LIN {X 0,Y 531.634,Z 644.42,A -85,B 0,C 180,E1 -4424.547,E2 -4424.547} C_VEL
LIN {X 0,Y 532.056,Z 633.262,A -85,B 0,C 180,E1 -4425.908,E2 -4425.908} C_VEL
LIN {X 0,Y 532.532,Z 621.032,A -85,B 0,C 180,E1 -4427.175,E2 -4427.175} C_VEL
LIN {X 0,Y 533.095,Z 607.731,A -85,B 0,C 180,E1 -4428.341,E2 -4428.341} C_VEL
LIN {X 0,Y 533.678,Z 593.146,A -85,B 0,C 180,E1 -4429.421,E2 -4429.421} C_VEL
LIN {X 0,Y 534.172,Z 578.934,A -85,B 0,C 180,E1 -4430.304,E2 -4430.304} C_VEL
LIN {X 0,Y 534.817,Z 563.436,A -85,B 0,C 180,E1 -4431.092,E2 -4431.092} C_VEL
LIN {X 0,Y 535.239,Z 549.202,A -85,B 0,C 180,E1 -4431.672,E2 -4431.672} C_VEL
LIN {X 0,Y 535.654,Z 532.786,A -85,B 0,C 180,E1 -4432.186,E2 -4432.186} C_VEL
LIN {X 0,Y 535.928,Z 517.434,A -85,B 0,C 180,E1 -4432.53,E2 -4432.53} C_VEL
LIN {X 0,Y 537.327,Z 326.241,A -85,B 0,C 180,E1 -4435.221,E2 -4435.221} C_VEL
LIN {X 0,Y 536.874,Z 322.172,A -85,B 0,C 180,E1 -4435.302,E2 -4435.302} C_VEL
LIN {X 0,Y 534.828,Z 310.98,A -85,B 0,C 180,E1 -4435.587,E2 -4435.587} C_VEL
LIN {X 0,Y 535.649,Z 284.434,A -85,B 0,C 180,E1 -4438.055,E2 -4438.055} C_VEL
LIN {X 0,Y 530.979,Z 268.658,A -85,B 0,C 180,E1 -4439.867,E2 -4439.867} C_VEL
LIN {X 0,Y 530.965,Z 268.659,A -85,B 0,C 180,E1 -4442.866,E2 -4442.866} C_VEL
LIN {X 0,Y 530.952,Z 268.661,A -85,B 0,C 180,E1 -4445.62,E2 -4445.62} C_VEL
LIN {X 0,Y 530.966,Z 268.656,A -85,B 0,C 180,E1 -4448.654,E2 -4448.654} C_VEL
LIN {X 0,Y 530.997,Z 268.657,A -85,B 0,C 180,E1 -4451.435,E2 -4451.435} C_VEL
LIN {X 0,Y 530.986,Z 268.651,A -85,B 0,C 180,E1 -4454.547,E2 -4454.547} C_VEL
LIN {X 0,Y 530.985,Z 268.65,A -85,B 0,C 180,E1 -4457.834,E2 -4457.834} C_VEL
LIN {X 0,Y 530.985,Z 268.65,A -85,B 0,C 180,E1 -4460.557,E2 -4460.557} C_VEL
LIN {X 0,Y 530.963,Z 268.658,A -85,B 0,C 180,E1 -4463.442,E2 -4463.442} C_VEL
LIN {X 0,Y 530.996,Z 268.65,A -85,B 0,C 180,E1 -4466.494,E2 -4466.494} C_VEL
LIN {X 0,Y 530.971,Z 268.658,A -85,B 0,C 180,E1 -4469.355,E2 -4469.355} C_VEL
LIN {X 0,Y 531.009,Z 268.648,A -85,B 0,C 180,E1 -4472.468,E2 -4472.468} C_VEL
LIN {X 0,Y 531.003,Z 268.655,A -85,B 0,C 180,E1 -4474.943,E2 -4474.943} C_VEL
LIN {X 0,Y 530.969,Z 268.652,A -85,B 0,C 180,E1 -4478.247,E2 -4478.247} C_VEL
LIN {X 0,Y 530.99,Z 268.645,A -85,B 0,C 180,E1 -4480.677,E2 -4480.677} C_VEL
LIN {X 0,Y 530.983,Z 268.659,A -85,B 0,C 180,E1 -4483.071,E2 -4483.071} C_VEL
LIN {X 0,Y 531.016,Z 268.644,A -85,B 0,C 180,E1 -4485.436,E2 -4485.436} C_VEL
LIN {X 0,Y 531.034,Z 268.644,A -85,B 0,C 180,E1 -4488.55,E2 -4488.55} C_VEL
LIN {X 0,Y 531.053,Z 268.641,A -85,B 0,C 180,E1 -4491.63,E2 -4491.63} C_VEL
LIN {X 0,Y 531.122,Z 268.63,A -85,B 0,C 180,E1 -4494.685,E2 -4494.685} C_VEL
LIN {X 0,Y 531.139,Z 268.632,A -85,B 0,C 180,E1 -4497.725,E2 -4497.725} C_VEL
LIN {X 0,Y 531.15,Z 268.628,A -85,B 0,C 180,E1 -4500.758,E2 -4500.758} C_VEL
LIN {X 0,Y 531.103,Z 268.641,A -85,B 0,C 180,E1 -4503.034,E2 -4503.034} C_VEL
LIN {X 0,Y 531.073,Z 268.638,A -85,B 0,C 180,E1 -4506.077,E2 -4506.077} C_VEL
LIN {X 0,Y 531.053,Z 268.634,A -85,B 0,C 180,E1 -4508.371,E2 -4508.371} C_VEL
LIN {X 0,Y 531.049,Z 268.644,A -85,B 0,C 180,E1 -4511.672,E2 -4511.672} C_VEL
LIN {X 0,Y 531.029,Z 268.645,A -85,B 0,C 180,E1 -4514.956,E2 -4514.956} C_VEL
LIN {X 0,Y 531.015,Z 268.647,A -85,B 0,C 180,E1 -4517.723,E2 -4517.723} C_VEL
LIN {X 0,Y 530.998,Z 268.65,A -85,B 0,C 180,E1 -4520.938,E2 -4520.938} C_VEL
LIN {X 0,Y 530.978,Z 268.652,A -85,B 0,C 180,E1 -4524.225,E2 -4524.225} C_VEL
LIN {X 0,Y 530.999,Z 268.655,A -85,B 0,C 180,E1 -4526.744,E2 -4526.744} C_VEL
LIN {X 0,Y 530.98,Z 268.655,A -85,B 0,C 180,E1 -4529.323,E2 -4529.323} C_VEL
LIN {X 0,Y 530.963,Z 268.653,A -85,B 0,C 180,E1 -4532.1,E2 -4532.1} C_VEL
LIN {X 0,Y 530.988,Z 268.657,A -85,B 0,C 180,E1 -4534.854,E2 -4534.854} C_VEL
LIN {X 0,Y 530.965,Z 268.649,A -85,B 0,C 180,E1 -4537.508,E2 -4537.508} C_VEL
LIN {X 0,Y 530.98,Z 268.654,A -85,B 0,C 180,E1 -4540.433,E2 -4540.433} C_VEL
LIN {X 0,Y 530.964,Z 268.655,A -85,B 0,C 180,E1 -4543.495,E2 -4543.495} C_VEL
LIN {X 0,Y 530.961,Z 268.655,A -85,B 0,C 180,E1 -4543.559,E2 -4543.559} C_VEL
LIN {X 0,Y 530.288,Z 268.74,A -85,B 0,C 180,E1 -4544.193,E2 -4544.193} C_VEL
LIN {X 0,Y 527.439,Z 269.098,A -85,B 0,C 180,E1 -4545.222,E2 -4545.222} C_VEL
LIN {X 0,Y 525.036,Z 269.401,A -85,B 0,C 180,E1 -4546.05,E2 -4546.05} C_VEL
LIN {X 0,Y 524.003,Z 269.527,A -85,B 0,C 180,E1 -4546.69,E2 -4546.69} C_VEL
LIN {X 0,Y 523.919,Z 269.536,A -85,B 0,C 180,E1 -4546.906,E2 -4546.906} C_VEL
LIN {X 0,Y 523.937,Z 269.53,A -85,B 0,C 180,E1 -4549.87,E2 -4549.87} C_VEL
LIN {X 0,Y 523.906,Z 269.529,A -85,B 0,C 180,E1 -4552.868,E2 -4552.868} C_VEL
LIN {X 0,Y 523.932,Z 269.53,A -85,B 0,C 180,E1 -4555.71,E2 -4555.71} C_VEL
LIN {X 0,Y 523.921,Z 269.537,A -85,B 0,C 180,E1 -4558.456,E2 -4558.456} C_VEL
LIN {X 0,Y 523.93,Z 269.538,A -85,B 0,C 180,E1 -4561.125,E2 -4561.125} C_VEL
LIN {X 0,Y 523.992,Z 269.628,A -85,B 0,C 180,E1 -4562.312,E2 -4562.312} C_VEL
LIN {X 0,Y 527.994,Z 284.16,A -85,B 0,C 180,E1 -4564.139,E2 -4564.139} C_VEL
LIN {X 0,Y 530.797,Z 296.653,A -85,B 0,C 180,E1 -4564.471,E2 -4564.471} C_VEL
LIN {X 0,Y 531.002,Z 300.708,A -85,B 0,C 180,E1 -4564.541,E2 -4564.541} C_VEL
LIN {X 0,Y 529.519,Z 486.107,A -85,B 0,C 180,E1 -4567.182,E2 -4567.182} C_VEL
LIN {X 0,Y 529.204,Z 502.429,A -85,B 0,C 180,E1 -4567.529,E2 -4567.529} C_VEL
LIN {X 0,Y 528.801,Z 517.915,A -85,B 0,C 180,E1 -4567.999,E2 -4567.999} C_VEL
LIN {X 0,Y 528.268,Z 533.513,A -85,B 0,C 180,E1 -4568.634,E2 -4568.634} C_VEL
LIN {X 0,Y 527.73,Z 547.349,A -85,B 0,C 180,E1 -4569.335,E2 -4569.335} C_VEL
LIN {X 0,Y 527.128,Z 561.913,A -85,B 0,C 180,E1 -4570.226,E2 -4570.226} C_VEL
LIN {X 0,Y 526.54,Z 575.392,A -85,B 0,C 180,E1 -4571.216,E2 -4571.216} C_VEL
LIN {X 0,Y 525.914,Z 587.91,A -85,B 0,C 180,E1 -4572.301,E2 -4572.301} C_VEL
LIN {X 0,Y 525.35,Z 599.656,A -85,B 0,C 180,E1 -4573.484,E2 -4573.484} C_VEL
LIN {X 0,Y 524.813,Z 610.629,A -85,B 0,C 180,E1 -4574.768,E2 -4574.768} C_VEL
LIN {X 0,Y 524.367,Z 621.269,A -85,B 0,C 180,E1 -4576.237,E2 -4576.237} C_VEL
LIN {X 0,Y 524.023,Z 630.883,A -85,B 0,C 180,E1 -4577.806,E2 -4577.806} C_VEL
LIN {X 0,Y 523.794,Z 638.055,A -85,B 0,C 180,E1 -4579.173,E2 -4579.173} C_VEL
LIN {X 0,Y 523.57,Z 644.914,A -85,B 0,C 180,E1 -4580.731,E2 -4580.731} C_VEL
LIN {X 0,Y 523.473,Z 650.575,A -85,B 0,C 180,E1 -4582.284,E2 -4582.284} C_VEL
LIN {X 0,Y 523.412,Z 655.13,A -85,B 0,C 180,E1 -4583.834,E2 -4583.834} C_VEL
LIN {X 0,Y 523.314,Z 658.548,A -85,B 0,C 180,E1 -4585.378,E2 -4585.378} C_VEL
LIN {X 0,Y 523.354,Z 661.03,A -85,B 0,C 180,E1 -4586.921,E2 -4586.921} C_VEL
LIN {X 0,Y 523.27,Z 662.449,A -85,B 0,C 180,E1 -4588.461,E2 -4588.461} C_VEL
LIN {X 0,Y 523.243,Z 662.997,A -85,B 0,C 180,E1 -4590,E2 -4590} C_VEL
LIN {X 0,Y 523.268,Z 662.506,A -85,B 0,C 180,E1 -4591.539,E2 -4591.539} C_VEL
LIN {X 0,Y 523.355,Z 661.143,A -85,B 0,C 180,E1 -4593.079,E2 -4593.079} C_VEL
LIN {X 0,Y 523.311,Z 658.718,A -85,B 0,C 180,E1 -4594.622,E2 -4594.622} C_VEL
LIN {X 0,Y 523.413,Z 655.368,A -85,B 0,C 180,E1 -4596.166,E2 -4596.166} C_VEL
LIN {X 0,Y 523.505,Z 649.617,A -85,B 0,C 180,E1 -4598.103,E2 -4598.103} C_VEL
LIN {X 0,Y 523.655,Z 642.056,A -85,B 0,C 180,E1 -4600.048,E2 -4600.048} C_VEL
LIN {X 0,Y 523.958,Z 634.003,A -85,B 0,C 180,E1 -4601.715,E2 -4601.715} C_VEL
LIN {X 0,Y 524.207,Z 625.622,A -85,B 0,C 180,E1 -4603.174,E2 -4603.174} C_VEL
LIN {X 0,Y 524.675,Z 614.98,A -85,B 0,C 180,E1 -4604.744,E2 -4604.744} C_VEL
LIN {X 0,Y 525.141,Z 603.993,A -85,B 0,C 180,E1 -4606.123,E2 -4606.123} C_VEL
LIN {X 0,Y 525.748,Z 590.982,A -85,B 0,C 180,E1 -4607.504,E2 -4607.504} C_VEL
LIN {X 0,Y 526.388,Z 577.69,A -85,B 0,C 180,E1 -4608.689,E2 -4608.689} C_VEL
LIN {X 0,Y 527.004,Z 564.595,A -85,B 0,C 180,E1 -4609.677,E2 -4609.677} C_VEL
LIN {X 0,Y 527.607,Z 550.668,A -85,B 0,C 180,E1 -4610.568,E2 -4610.568} C_VEL
LIN {X 0,Y 528.178,Z 536.055,A -85,B 0,C 180,E1 -4611.341,E2 -4611.341} C_VEL
LIN {X 0,Y 528.668,Z 521.497,A -85,B 0,C 180,E1 -4611.955,E2 -4611.955} C_VEL
LIN {X 0,Y 529.106,Z 504.71,A -85,B 0,C 180,E1 -4612.501,E2 -4612.501} C_VEL
LIN {X 0,Y 529.47,Z 488.35,A -85,B 0,C 180,E1 -4612.871,E2 -4612.871} C_VEL
LIN {X 0,Y 531.006,Z 298.489,A -85,B 0,C 180,E1 -4615.581,E2 -4615.581} C_VEL
LIN {X 0,Y 528.356,Z 285.26,A -85,B 0,C 180,E1 -4615.916,E2 -4615.916} C_VEL
LIN {X 0,Y 527.894,Z 283.813,A -85,B 0,C 180,E1 -4615.979,E2 -4615.979} C_VEL
LIN {X 0,Y 523.963,Z 269.532,A -85,B 0,C 180,E1 -4617.819,E2 -4617.819} C_VEL
LIN {X 0,Y 523.944,Z 269.534,A -85,B 0,C 180,E1 -4620.854,E2 -4620.854} C_VEL
LIN {X 0,Y 523.958,Z 269.533,A -85,B 0,C 180,E1 -4623.734,E2 -4623.734} C_VEL
LIN {X 0,Y 523.897,Z 269.529,A -85,B 0,C 180,E1 -4626.4,E2 -4626.4} C_VEL
LIN {X 0,Y 523.918,Z 269.539,A -85,B 0,C 180,E1 -4629.085,E2 -4629.085} C_VEL
LIN {X 0,Y 523.951,Z 269.526,A -85,B 0,C 180,E1 -4632.119,E2 -4632.119} C_VEL
LIN {X 0,Y 523.953,Z 269.531,A -85,B 0,C 180,E1 -4635.309,E2 -4635.309} C_VEL
LIN {X 0,Y 523.956,Z 269.528,A -85,B 0,C 180,E1 -4638.689,E2 -4638.689} C_VEL
LIN {X 0,Y 523.915,Z 269.539,A -85,B 0,C 180,E1 -4641.08,E2 -4641.08} C_VEL
LIN {X 0,Y 523.922,Z 269.531,A -85,B 0,C 180,E1 -4643.827,E2 -4643.827} C_VEL
LIN {X 0,Y 523.939,Z 269.53,A -85,B 0,C 180,E1 -4646.635,E2 -4646.635} C_VEL
LIN {X 0,Y 523.953,Z 269.534,A -85,B 0,C 180,E1 -4649.355,E2 -4649.355} C_VEL
LIN {X 0,Y 523.974,Z 269.519,A -85,B 0,C 180,E1 -4652.281,E2 -4652.281} C_VEL
LIN {X 0,Y 523.95,Z 269.529,A -85,B 0,C 180,E1 -4654.581,E2 -4654.581} C_VEL
LIN {X 0,Y 523.914,Z 269.533,A -85,B 0,C 180,E1 -4657.107,E2 -4657.107} C_VEL
LIN {X 0,Y 523.976,Z 269.524,A -85,B 0,C 180,E1 -4659.866,E2 -4659.866} C_VEL
LIN {X 0,Y 523.964,Z 269.53,A -85,B 0,C 180,E1 -4662.837,E2 -4662.837} C_VEL
LIN {X 0,Y 523.974,Z 269.529,A -85,B 0,C 180,E1 -4665.236,E2 -4665.236} C_VEL
LIN {X 0,Y 524.01,Z 269.52,A -85,B 0,C 180,E1 -4668.394,E2 -4668.394} C_VEL
LIN {X 0,Y 523.998,Z 269.521,A -85,B 0,C 180,E1 -4671.516,E2 -4671.516} C_VEL
LIN {X 0,Y 524.083,Z 269.514,A -85,B 0,C 180,E1 -4674.614,E2 -4674.614} C_VEL
LIN {X 0,Y 524.11,Z 269.502,A -85,B 0,C 180,E1 -4677.694,E2 -4677.694} C_VEL
LIN {X 0,Y 524.12,Z 269.512,A -85,B 0,C 180,E1 -4680.768,E2 -4680.768} C_VEL
LIN {X 0,Y 524.069,Z 269.511,A -85,B 0,C 180,E1 -4683.075,E2 -4683.075} C_VEL
LIN {X 0,Y 524.05,Z 269.514,A -85,B 0,C 180,E1 -4686.159,E2 -4686.159} C_VEL
LIN {X 0,Y 523.994,Z 269.52,A -85,B 0,C 180,E1 -4689.262,E2 -4689.262} C_VEL
LIN {X 0,Y 524,Z 269.519,A -85,B 0,C 180,E1 -4691.739,E2 -4691.739} C_VEL
LIN {X 0,Y 523.99,Z 269.528,A -85,B 0,C 180,E1 -4695.052,E2 -4695.052} C_VEL
LIN {X 0,Y 523.961,Z 269.525,A -85,B 0,C 180,E1 -4697.969,E2 -4697.969} C_VEL
LIN {X 0,Y 523.969,Z 269.528,A -85,B 0,C 180,E1 -4700.41,E2 -4700.41} C_VEL
LIN {X 0,Y 523.914,Z 269.542,A -85,B 0,C 180,E1 -4702.893,E2 -4702.893} C_VEL
LIN {X 0,Y 523.949,Z 269.531,A -85,B 0,C 180,E1 -4705.419,E2 -4705.419} C_VEL
LIN {X 0,Y 523.964,Z 269.527,A -85,B 0,C 180,E1 -4707.999,E2 -4707.999} C_VEL
LIN {X 0,Y 523.941,Z 269.538,A -85,B 0,C 180,E1 -4710.855,E2 -4710.855} C_VEL
LIN {X 0,Y 523.958,Z 269.528,A -85,B 0,C 180,E1 -4713.735,E2 -4713.735} C_VEL
LIN {X 0,Y 523.92,Z 269.535,A -85,B 0,C 180,E1 -4716.404,E2 -4716.404} C_VEL
LIN {X 0,Y 523.918,Z 269.538,A -85,B 0,C 180,E1 -4719.085,E2 -4719.085} C_VEL
LIN {X 0,Y 523.954,Z 269.53,A -85,B 0,C 180,E1 -4722.118,E2 -4722.118} C_VEL
LIN {X 0,Y 523.953,Z 269.53,A -85,B 0,C 180,E1 -4725.309,E2 -4725.309} C_VEL
LIN {X 0,Y 523.959,Z 269.535,A -85,B 0,C 180,E1 -4728.689,E2 -4728.689} C_VEL
LIN {X 0,Y 523.913,Z 269.534,A -85,B 0,C 180,E1 -4731.898,E2 -4731.898} C_VEL
LIN {X 0,Y 523.922,Z 269.53,A -85,B 0,C 180,E1 -4734.911,E2 -4734.911} C_VEL
LIN {X 0,Y 523.933,Z 269.532,A -85,B 0,C 180,E1 -4737.68,E2 -4737.68} C_VEL
LIN {X 0,Y 523.952,Z 269.618,A -85,B 0,C 180,E1 -4739.829,E2 -4739.829} C_VEL
LIN {X 0,Y 529.028,Z 286.983,A -85,B 0,C 180,E1 -4741.828,E2 -4741.828} C_VEL
LIN {X 0,Y 528.165,Z 310.972,A -85,B 0,C 180,E1 -4744.086,E2 -4744.086} C_VEL
LIN {X 0,Y 530.903,Z 326.3,A -85,B 0,C 180,E1 -4744.456,E2 -4744.456} C_VEL
LIN {X 0,Y 529.373,Z 517.228,A -85,B 0,C 180,E1 -4747.176,E2 -4747.176} C_VEL
LIN {X 0,Y 529.093,Z 532.575,A -85,B 0,C 180,E1 -4747.524,E2 -4747.524} C_VEL
LIN {X 0,Y 528.577,Z 548.991,A -85,B 0,C 180,E1 -4748.041,E2 -4748.041} C_VEL
LIN {X 0,Y 528.149,Z 564.056,A -85,B 0,C 180,E1 -4748.666,E2 -4748.666} C_VEL
LIN {X 0,Y 527.395,Z 580.505,A -85,B 0,C 180,E1 -4749.525,E2 -4749.525} C_VEL
LIN {X 0,Y 526.761,Z 595.805,A -85,B 0,C 180,E1 -4750.516,E2 -4750.516} C_VEL
LIN {X 0,Y 526.188,Z 608.537,A -85,B 0,C 180,E1 -4751.496,E2 -4751.496} C_VEL
LIN {X 0,Y 525.602,Z 621.805,A -85,B 0,C 180,E1 -4752.692,E2 -4752.692} C_VEL
LIN {X 0,Y 525.098,Z 633.053,A -85,B 0,C 180,E1 -4753.876,E2 -4753.876} C_VEL
LIN {X 0,Y 524.654,Z 644.274,A -85,B 0,C 180,E1 -4755.255,E2 -4755.255} C_VEL
LIN {X 0,Y 524.176,Z 655.148,A -85,B 0,C 180,E1 -4756.825,E2 -4756.825} C_VEL
LIN {X 0,Y 523.934,Z 664.267,A -85,B 0,C 180,E1 -4758.392,E2 -4758.392} C_VEL
LIN {X 0,Y 523.658,Z 671.855,A -85,B 0,C 180,E1 -4759.952,E2 -4759.952} C_VEL
LIN {X 0,Y 523.503,Z 679.465,A -85,B 0,C 180,E1 -4761.897,E2 -4761.897} C_VEL
LIN {X 0,Y 523.411,Z 685.25,A -85,B 0,C 180,E1 -4763.834,E2 -4763.834} C_VEL
LIN {X 0,Y 523.312,Z 688.633,A -85,B 0,C 180,E1 -4765.378,E2 -4765.378} C_VEL
LIN {X 0,Y 523.353,Z 691.091,A -85,B 0,C 180,E1 -4766.921,E2 -4766.921} C_VEL
LIN {X 0,Y 523.268,Z 692.478,A -85,B 0,C 180,E1 -4768.461,E2 -4768.461} C_VEL
LIN {X 0,Y 523.242,Z 693,A -85,B 0,C 180,E1 -4770,E2 -4770} C_VEL
LIN {X 0,Y 523.268,Z 692.477,A -85,B 0,C 180,E1 -4771.539,E2 -4771.539} C_VEL
LIN {X 0,Y 523.353,Z 691.089,A -85,B 0,C 180,E1 -4773.079,E2 -4773.079} C_VEL
LIN {X 0,Y 523.312,Z 688.633,A -85,B 0,C 180,E1 -4774.622,E2 -4774.622} C_VEL
LIN {X 0,Y 523.411,Z 685.253,A -85,B 0,C 180,E1 -4776.167,E2 -4776.167} C_VEL
LIN {X 0,Y 523.503,Z 679.467,A -85,B 0,C 180,E1 -4778.103,E2 -4778.103} C_VEL
LIN {X 0,Y 523.658,Z 671.855,A -85,B 0,C 180,E1 -4780.048,E2 -4780.048} C_VEL
LIN {X 0,Y 523.956,Z 663.711,A -85,B 0,C 180,E1 -4781.715,E2 -4781.715} C_VEL
LIN {X 0,Y 524.176,Z 655.149,A -85,B 0,C 180,E1 -4783.175,E2 -4783.175} C_VEL
LIN {X 0,Y 524.649,Z 644.275,A -85,B 0,C 180,E1 -4784.745,E2 -4784.745} C_VEL
LIN {X 0,Y 525.098,Z 633.05,A -85,B 0,C 180,E1 -4786.124,E2 -4786.124} C_VEL
LIN {X 0,Y 525.666,Z 620.822,A -85,B 0,C 180,E1 -4787.406,E2 -4787.406} C_VEL
